KUKA KRL program: MyProgram_091().src

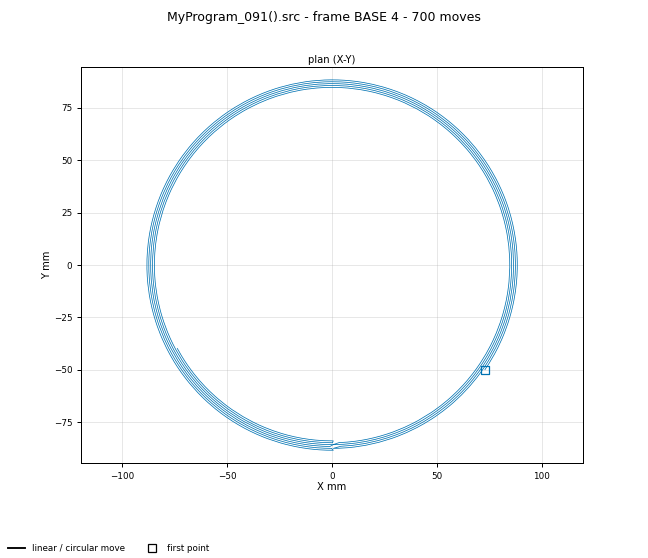
[picture p0: tool path of MyProgram_091().src in frame BASE 4, 700 of 700 moves have a stored position in this frame; points joined in program order, loops and branches not executed]
&ACCESS RVP
&REL 1
&PARAM TEMPLATE = C:\KRC\Roboter\Template\vorgabe
&PARAM EDITMASK = *
DEF MyProgram_091()
; ---- Setting reference (Base) ----
$BASE = BASE_DATA[4]

; --------------------------
; ---- Setting tool (TCP) ----
$TOOL = TOOL_DATA[3]
; --------------------------

$VEL.CP = VEL_APROX_PRINT
Startdeposition()
$VEL.CP = VEL_PRINT
LIN {X 72.876,Y -49.889,Z 87,A -38.6628,B 24.9212,C -2.0494,E1 25.1329,E2 483.5993} C_DIS
LIN {X 74.7508,Y -47.0321,Z 87,A -36.5976,B 24.9212,C -2.0503,E1 25.136,E2 481.5424} C_DIS
LIN {X 77.4491,Y -42.4429,Z 87,A -33.0497,B 24.9201,C -2.0636,E1 25.141,E2 477.9815} C_DIS
LIN {X 79.025,Y -39.4299,Z 87,A -30.5206,B 24.9187,C -2.0816,E1 25.1442,E2 475.4232} C_DIS
LIN {X 80.9108,Y -35.3988,Z 87,A -27.9647,B 24.919,C -2.0785,E1 25.1471,E2 472.8887} C_DIS
LIN {X 82.1401,Y -32.4446,Z 87,A -25.9813,B 24.9187,C -2.0815,E1 25.1492,E2 470.9091} C_DIS
LIN {X 83.9091,Y -27.5504,Z 87,A -22.6052,B 24.9179,C -2.0919,E1 25.1523,E2 467.5274} C_DIS
LIN {X 84.8703,Y -24.4292,Z 87,A -20.491,B 24.9174,C -2.0984,E1 25.154,E2 465.41} C_DIS
LIN {X 85.5175,Y -22.0541,Z 87,A -18.418,B 24.9157,C -2.1205,E1 25.1555,E2 463.2967} C_DIS
LIN {X 86.2783,Y -18.8591,Z 87,A -16.8201,B 24.9167,C -2.1081,E1 25.1564,E2 461.7374} C_DIS
LIN {X 86.7492,Y -16.5591,Z 87,A -15.0502,B 24.9156,C -2.1218,E1 25.1574,E2 459.9455} C_DIS
LIN {X 87.4227,Y -12.5256,Z 87,A -12.6764,B 24.9156,C -2.1203,E1 25.1584,E2 457.5893} C_DIS
LIN {X 87.8803,Y -8.7666,Z 87,A -10.1907,B 24.915,C -2.1292,E1 25.1591,E2 455.0972} C_DIS
LIN {X 88.1529,Y -5.3772,Z 87,A -7.9487,B 24.9143,C -2.1375,E1 25.1596,E2 452.8488} C_DIS
LIN {X 88.2975,Y -1.7856,Z 87,A -5.7756,B 24.9142,C -2.1393,E1 25.1598,E2 450.6844} C_DIS
LIN {X 88.3023,Y 1.525,Z 87,A -3.8298,B 24.9142,C -2.139,E1 25.1598,E2 448.751} C_DIS
LIN {X 88.2492,Y 3.4377,Z 87,A -2.4189,B 24.9134,C -2.149,E1 25.1596,E2 447.3249} C_DIS
LIN {X 88.101,Y 6.1542,Z 87,A -0.5423,B 24.9126,C -2.1586,E1 25.1593,E2 445.4368} C_DIS
LIN {X 87.7851,Y 9.6757,Z 87,A 1.7717,B 24.912,C -2.1666,E1 25.1586,E2 443.1177} C_DIS
LIN {X 87.4539,Y 12.306,Z 87,A 3.3765,B 24.9118,C -2.1679,E1 25.158,E2 441.5192} C_DIS
LIN {X 86.9147,Y 15.667,Z 87,A 6.3248,B 24.9091,C -2.2013,E1 25.1566,E2 438.5094} C_DIS
LIN {X 86.0978,Y 19.6679,Z 87,A 8.2385,B 24.9106,C -2.1831,E1 25.1554,E2 436.6497} C_DIS
LIN {X 85.2224,Y 23.1685,Z 87,A 11.3311,B 24.9078,C -2.217,E1 25.1532,E2 433.4948} C_DIS
LIN {X 84.0146,Y 27.2242,Z 87,A 13.1855,B 24.9098,C -2.1935,E1 25.1517,E2 431.7066} C_DIS
LIN {X 82.9978,Y 30.1827,Z 87,A 14.9428,B 24.9101,C -2.1898,E1 25.15,E2 429.9677} C_DIS
LIN {X 81.9785,Y 32.8537,Z 87,A 17.2118,B 24.9084,C -2.2098,E1 25.1477,E2 427.6642} C_DIS
LIN {X 80.5997,Y 36.1019,Z 87,A 19.3758,B 24.9082,C -2.2119,E1 25.1453,E2 425.507} C_DIS
LIN {X 79.2608,Y 38.9542,Z 87,A 21.315,B 24.9081,C -2.2139,E1 25.143,E2 423.5735} C_DIS
LIN {X 77.959,Y 41.4989,Z 87,A 23.2226,B 24.9075,C -2.2209,E1 25.1405,E2 421.6595} C_DIS
LIN {X 76.1764,Y 44.6862,Z 87,A 25.6641,B 24.9067,C -2.2298,E1 25.1371,E2 419.2097} C_DIS
LIN {X 74.6097,Y 47.2577,Z 87,A 27.6005,B 24.9064,C -2.2342,E1 25.1342,E2 417.2726} C_DIS
LIN {X 72.7642,Y 50.0518,Z 87,A 29.7426,B 24.906,C -2.2387,E1 25.1309,E2 415.1305} C_DIS
LIN {X 70.4422,Y 53.269,Z 87,A 32.3068,B 24.9055,C -2.2447,E1 25.1267,E2 412.5645} C_DIS
LIN {X 68.1897,Y 56.1245,Z 87,A 34.6943,B 24.9049,C -2.2512,E1 25.1225,E2 410.1727} C_DIS
LIN {X 64.9745,Y 59.816,Z 87,A 37.8698,B 24.9043,C -2.2584,E1 25.1166,E2 406.9945} C_DIS
LIN {X 62.6446,Y 62.2522,Z 87,A 39.9936,B 24.9041,C -2.2609,E1 25.1124,E2 404.8738} C_DIS
LIN {X 60.3809,Y 64.4499,Z 87,A 42.1613,B 24.9034,C -2.2692,E1 25.108,E2 402.6953} C_DIS
LIN {X 57.7117,Y 66.8523,Z 87,A 44.4118,B 24.9032,C -2.2711,E1 25.1033,E2 400.4494} C_DIS
LIN {X 55.9301,Y 68.3492,Z 87,A 46.0715,B 24.9026,C -2.279,E1 25.0997,E2 398.7771} C_DIS
LIN {X 52.7405,Y 70.8393,Z 87,A 48.5236,B 24.9026,C -2.2778,E1 25.0943,E2 396.3369} C_DIS
LIN {X 49.8742,Y 72.886,Z 87,A 50.7541,B 24.9025,C -2.2797,E1 25.0892,E2 394.1095} C_DIS
LIN {X 47.2166,Y 74.6354,Z 87,A 52.8049,B 24.9023,C -2.2825,E1 25.0844,E2 392.0588} C_DIS
LIN {X 44.6136,Y 76.2193,Z 87,A 54.8992,B 24.9017,C -2.2894,E1 25.0793,E2 389.9547} C_DIS
LIN {X 40.7584,Y 78.349,Z 87,A 57.6799,B 24.9016,C -2.2906,E1 25.0725,E2 387.179} C_DIS
LIN {X 37.7561,Y 79.8391,Z 87,A 59.8219,B 24.9014,C -2.2922,E1 25.0671,E2 385.0389} C_DIS
LIN {X 34.8344,Y 81.1568,Z 87,A 61.9798,B 24.901,C -2.2971,E1 25.0616,E2 382.8748} C_DIS
LIN {X 31.3951,Y 82.5468,Z 87,A 64.2661,B 24.9011,C -2.2954,E1 25.0556,E2 380.5973} C_DIS
LIN {X 27.7885,Y 83.8309,Z 87,A 66.9063,B 24.9005,C -2.3027,E1 25.0486,E2 377.945} C_DIS
LIN {X 24.1511,Y 84.9491,Z 87,A 69.3497,B 24.9005,C -2.3037,E1 25.0421,E2 375.5036} C_DIS
LIN {X 19.3333,Y 86.1749,Z 87,A 72.7743,B 24.8997,C -2.3119,E1 25.0328,E2 372.0643} C_DIS
LIN {X 15.0004,Y 87.0333,Z 87,A 75.3209,B 24.9005,C -2.3027,E1 25.0258,E2 369.5426} C_DIS
LIN {X 11.7786,Y 87.5275,Z 87,A 77.488,B 24.9003,C -2.3049,E1 25.0198,E2 367.3721} C_DIS
LIN {X 8.3793,Y 87.9174,Z 87,A 79.6385,B 24.9005,C -2.303,E1 25.0139,E2 365.2275} C_DIS
LIN {X 5.8507,Y 88.1215,Z 87,A 81.1313,B 24.9009,C -2.2981,E1 25.0098,E2 363.7469} C_DIS
LIN {X 2.8316,Y 88.2701,Z 87,A 83.2135,B 24.9006,C -2.3019,E1 25.0039,E2 361.6564} C_DIS
LIN {X -0.4871,Y 88.3141,Z 87,A 85.3405,B 24.9006,C -2.3007,E1 24.998,E2 359.5324} C_DIS
LIN {X -3.58,Y 88.2431,Z 87,A 87.5251,B 24.9003,C -2.3057,E1 24.9919,E2 357.3356} C_DIS
LIN {X -9.587,Y 87.7944,Z 87,A 91.3179,B 24.9007,C -2.3002,E1 24.9814,E2 353.5541} C_DIS
LIN {X -12.8181,Y 87.3812,Z 87,A 93.176,B 24.9015,C -2.2909,E1 24.9763,E2 351.7167} C_DIS
LIN {X -19.1362,Y 86.2179,Z 87,A 98.0168,B 24.9,C -2.3085,E1 24.9629,E2 346.8286} C_DIS
LIN {X -24.8016,Y 84.762,Z 87,A 101.1149,B 24.9022,C -2.283,E1 24.9547,E2 343.7865} C_DIS
LIN {X -27.1803,Y 84.0288,Z 87,A 102.9141,B 24.9019,C -2.2868,E1 24.9498,E2 341.975} C_DIS
LIN {X -30.117,Y 83.0217,Z 87,A 104.987,B 24.9019,C -2.2861,E1 24.9444,E2 339.8997} C_DIS
LIN {X -33.1255,Y 81.8679,Z 87,A 107.1485,B 24.902,C -2.2855,E1 24.9387,E2 337.735} C_DIS
LIN {X -36.3766,Y 80.4759,Z 87,A 109.4796,B 24.9022,C -2.2832,E1 24.9328,E2 335.4037} C_DIS
LIN {X -39.1194,Y 79.1789,Z 87,A 111.3587,B 24.9027,C -2.2774,E1 24.9281,E2 333.5336} C_DIS
LIN {X -41.9795,Y 77.7004,Z 87,A 113.3448,B 24.9033,C -2.2709,E1 24.9232,E2 331.5577} C_DIS
LIN {X -46.5097,Y 75.0771,Z 87,A 116.9653,B 24.9033,C -2.2715,E1 24.9145,E2 327.9247} C_DIS
LIN {X -49.4678,Y 73.1612,Z 87,A 119.2238,B 24.9036,C -2.2663,E1 24.9092,E2 325.6712} C_DIS
LIN {X -52.1803,Y 71.2519,Z 87,A 121.7484,B 24.9031,C -2.2731,E1 24.9035,E2 323.1215} C_DIS
LIN {X -56.1307,Y 68.1845,Z 87,A 124.6939,B 24.9044,C -2.2571,E1 24.8971,E2 320.2031} C_DIS
LIN {X -58.7959,Y 65.899,Z 87,A 126.8822,B 24.9051,C -2.2494,E1 24.8925,E2 318.0248} C_DIS
LIN {X -61.1916,Y 63.6807,Z 87,A 129.2287,B 24.9049,C -2.2512,E1 24.8877,E2 315.6642} C_DIS
LIN {X -63.993,Y 60.8667,Z 87,A 131.6694,B 24.9058,C -2.2409,E1 24.883,E2 313.2375} C_DIS
LIN {X -66.1895,Y 58.4706,Z 87,A 133.8713,B 24.906,C -2.2384,E1 24.8789,E2 311.0319} C_DIS
LIN {X -68.3105,Y 55.9778,Z 87,A 136.0783,B 24.9063,C -2.2353,E1 24.8749,E2 308.8219} C_DIS
LIN {X -71.2925,Y 52.1248,Z 87,A 139.5827,B 24.9061,C -2.237,E1 24.869,E2 305.2966} C_DIS
LIN {X -73.1619,Y 49.4667,Z 87,A 141.0522,B 24.9082,C -2.2125,E1 24.8668,E2 303.8784} C_DIS
LIN {X -75.9695,Y 45.0363,Z 87,A 144.5868,B 24.9087,C -2.2067,E1 24.8616,E2 300.3396} C_DIS
LIN {X -77.3872,Y 42.557,Z 87,A 146.5252,B 24.9089,C -2.2038,E1 24.8589,E2 298.3979} C_DIS
LIN {X -78.8169,Y 39.8455,Z 87,A 148.6496,B 24.9091,C -2.202,E1 24.8562,E2 296.2666} C_DIS
LIN {X -80.4836,Y 36.3595,Z 87,A 150.9735,B 24.9101,C -2.1892,E1 24.8535,E2 293.9605} C_DIS
LIN {X -81.7261,Y 33.4739,Z 87,A 153.0561,B 24.9105,C -2.1843,E1 24.8512,E2 291.878} C_DIS
LIN {X -82.8825,Y 30.4988,Z 87,A 155.1598,B 24.9109,C -2.1789,E1 24.8492,E2 289.7753} C_DIS
LIN {X -83.9638,Y 27.3812,Z 87,A 157.4119,B 24.9112,C -2.1755,E1 24.8472,E2 287.5185} C_DIS
LIN {X -84.9579,Y 24.1201,Z 87,A 159.5991,B 24.9118,C -2.1679,E1 24.8454,E2 285.3368} C_DIS
LIN {X -85.7975,Y 20.9382,Z 87,A 161.6195,B 24.9127,C -2.1579,E1 24.8441,E2 283.3285} C_DIS
LIN {X -86.4497,Y 18.0599,Z 87,A 163.6354,B 24.9129,C -2.1547,E1 24.8429,E2 281.3083} C_DIS
LIN {X -87.0374,Y 14.9757,Z 87,A 165.6786,B 24.9134,C -2.1484,E1 24.8419,E2 279.268} C_DIS
LIN {X -87.5816,Y 11.3616,Z 87,A 168.9039,B 24.912,C -2.1657,E1 24.8407,E2 275.9822} C_DIS
LIN {X -88.0383,Y 6.9906,Z 87,A 171.1962,B 24.9141,C -2.1403,E1 24.8401,E2 273.7369} C_DIS
LIN {X -88.2709,Y 2.807,Z 87,A 173.5689,B 24.9156,C -2.1216,E1 24.8398,E2 271.3945} C_DIS
LIN {X -88.2983,Y -1.7412,Z 87,A 176.7792,B 24.9157,C -2.1197,E1 24.8398,E2 268.1695} C_DIS
LIN {X -88.1559,Y -5.3252,Z 87,A 178.975,B 24.9166,C -2.1084,E1 24.8402,E2 265.9872} C_DIS
LIN {X -87.8679,Y -8.8855,Z 87,A -178.2885,B 24.9162,C -2.1133,E1 24.8409,E2 263.2227} C_DIS
LIN {X -87.1817,Y -14.1128,Z 87,A -175.1401,B 24.9177,C -2.0947,E1 24.8422,E2 260.1} C_DIS
LIN {X -86.608,Y -17.2887,Z 87,A -173.0562,B 24.9182,C -2.0879,E1 24.8432,E2 258.02} C_DIS
LIN {X -85.8301,Y -20.8043,Z 87,A -170.8084,B 24.919,C -2.0782,E1 24.8447,E2 255.7821} C_DIS
LIN {X -85.1046,Y -23.6023,Z 87,A -168.8704,B 24.9193,C -2.0743,E1 24.8461,E2 253.8421} C_DIS
LIN {X -84.1569,Y -26.7844,Z 87,A -166.6296,B 24.9196,C -2.0704,E1 24.8479,E2 251.5977} C_DIS
LIN {X -83.3448,Y -29.2106,Z 87,A -164.2506,B 24.9183,C -2.0868,E1 24.8502,E2 249.1663} C_DIS
LIN {X -81.8433,Y -33.186,Z 87,A -162.2766,B 24.9208,C -2.0557,E1 24.8522,E2 247.2554} C_DIS
LIN {X -80.9152,Y -35.3886,Z 87,A -160.3188,B 24.9202,C -2.0632,E1 24.8544,E2 245.2687} C_DIS
LIN {X -79.0112,Y -39.4578,Z 87,A -157.8931,B 24.9219,C -2.0407,E1 24.8573,E2 242.8837} C_DIS
LIN {X -77.5103,Y -42.3301,Z 87,A -155.4738,B 24.9216,C -2.0443,E1 24.8605,E2 240.4428} C_DIS
LIN {X -75.5172,Y -45.7905,Z 87,A -153.1118,B 24.9227,C -2.0307,E1 24.8638,E2 238.1011} C_DIS
LIN {X -73.8148,Y -48.4873,Z 87,A -150.9893,B 24.923,C -2.027,E1 24.867,E2 235.9768} C_DIS
LIN {X -71.9019,Y -51.281,Z 87,A -148.6632,B 24.923,C -2.0254,E1 24.8708,E2 233.643} C_DIS
LIN {X -69.5864,Y -54.3836,Z 87,A -146.2279,B 24.9237,C -2.017,E1 24.8749,E2 231.2161} C_DIS
LIN {X -68.083,Y -56.2528,Z 87,A -144.2851,B 24.9231,C -2.0251,E1 24.8784,E2 229.2452} C_DIS
LIN {X -64.0638,Y -60.7914,Z 87,A -140.5474,B 24.9242,C -2.0104,E1 24.8854,E2 225.5258} C_DIS
LIN {X -61.2434,Y -63.6307,Z 87,A -138.2242,B 24.9252,C -1.9968,E1 24.8899,E2 223.2254} C_DIS
LIN {X -59.1443,Y -65.5871,Z 87,A -136.313,B 24.9254,C -1.9945,E1 24.8939,E2 221.3117} C_DIS
LIN {X -55.4752,Y -68.7179,Z 87,A -133.0922,B 24.9256,C -1.9914,E1 24.9008,E2 218.0859} C_DIS
LIN {X -52.8784,Y -70.7356,Z 87,A -130.9123,B 24.9258,C -1.9891,E1 24.9056,E2 215.9037} C_DIS
LIN {X -50.2741,Y -72.6096,Z 87,A -128.825,B 24.9261,C -1.9858,E1 24.9104,E2 213.817} C_DIS
LIN {X -47.5755,Y -74.4057,Z 87,A -126.707,B 24.9263,C -1.983,E1 24.9154,E2 211.6989} C_DIS
LIN {X -44.9756,Y -76.0053,Z 87,A -124.6208,B 24.9263,C -1.9834,E1 24.9204,E2 209.6053} C_DIS
LIN {X -41.6869,Y -77.8592,Z 87,A -122.2867,B 24.9268,C -1.9766,E1 24.9261,E2 207.2809} C_DIS
LIN {X -38.9012,Y -79.2871,Z 87,A -120.2764,B 24.927,C -1.9734,E1 24.9311,E2 205.2727} C_DIS
LIN {X -36.1322,Y -80.586,Z 87,A -118.266,B 24.927,C -1.972,E1 24.9362,E2 203.2607} C_DIS
LIN {X -32.7878,Y -82.0053,Z 87,A -115.8818,B 24.9272,C -1.9705,E1 24.9424,E2 200.8747} C_DIS
LIN {X -30.3038,Y -82.9536,Z 87,A -113.7469,B 24.9263,C -1.982,E1 24.948,E2 198.7082} C_DIS
LIN {X -24.4184,Y -84.8733,Z 87,A -110.1572,B 24.9276,C -1.9654,E1 24.9575,E2 195.1516} C_DIS
LIN {X -22.1968,Y -85.4808,Z 87,A -108.4317,B 24.9271,C -1.972,E1 24.9622,E2 193.4081} C_DIS
LIN {X -18.1313,Y -86.435,Z 87,A -106.0112,B 24.9279,C -1.9614,E1 24.9688,E2 191.0096} C_DIS
LIN {X -15.1651,Y -87.0049,Z 87,A -103.9211,B 24.9276,C -1.9649,E1 24.9745,E2 188.909} C_DIS
LIN {X -11.645,Y -87.5448,Z 87,A -101.7389,B 24.928,C -1.9603,E1 24.9805,E2 186.736} C_DIS
LIN {X -9.0148,Y -87.8543,Z 87,A -100.1645,B 24.9283,C -1.9554,E1 24.9849,E2 185.1722} C_DIS
LIN {X -6.1629,Y -88.1004,Z 87,A -98.1033,B 24.9278,C -1.962,E1 24.9907,E2 183.0945} C_DIS
LIN {X -2.6223,Y -88.2765,Z 87,A -95.8044,B 24.9278,C -1.9622,E1 24.9971,E2 180.7946} C_DIS
LIN {X 0.5878,Y -88.3126,Z 87,A -94.072,B 24.9286,C -1.9512,E1 25.0019,E2 179.0883} C_DIS
Enddeposition()
LIN {X 0.5878,Y -88.3126,Z 87,A -94.072,B 24.9286,C -1.9512,E1 25.0019,E2 179.0883} C_DIS
Startdeposition()
$VEL.CP = VEL_PRINT
LIN {X -0.2815,Y -87.4214,Z 87,A -95.3283,B 24.9291,C -1.9446,E1 24.9983,E2 180.3603} C_DIS
LIN {X -3.6833,Y -87.3438,Z 87,A -97.4905,B 24.929,C -1.9464,E1 24.9923,E2 182.5184} C_DIS
LIN {X -7.3441,Y -87.113,Z 87,A -100.0671,B 24.9294,C -1.941,E1 24.9851,E2 185.1089} C_DIS
LIN {X -10.6188,Y -86.7753,Z 87,A -102.1476,B 24.9292,C -1.9437,E1 24.9793,E2 187.1844} C_DIS
LIN {X -13.9854,Y -86.2966,Z 87,A -104.6701,B 24.9298,C -1.9351,E1 24.9723,E2 189.7295} C_DIS
LIN {X -18.097,Y -85.5294,Z 87,A -107.3335,B 24.9295,C -1.9386,E1 24.965,E2 192.3876} C_DIS
LIN {X -22.0017,Y -84.6079,Z 87,A -109.8167,B 24.9291,C -1.9446,E1 24.9583,E2 194.86} C_DIS
LIN {X -26.6799,Y -83.2511,Z 87,A -113.3252,B 24.9296,C -1.9372,E1 24.9489,E2 198.3922} C_DIS
LIN {X -30.4817,Y -81.9368,Z 87,A -115.7071,B 24.9289,C -1.9472,E1 24.9427,E2 200.755} C_DIS
LIN {X -35.5927,Y -79.8486,Z 87,A -118.9086,B 24.9277,C -1.9636,E1 24.9345,E2 203.9248} C_DIS
LIN {X -39.0234,Y -78.2287,Z 87,A -121.728,B 24.9282,C -1.9565,E1 24.9273,E2 206.7684} C_DIS
LIN {X -44.0876,Y -75.4917,Z 87,A -125.2495,B 24.9273,C -1.9691,E1 24.9188,E2 210.27} C_DIS
LIN {X -48.2363,Y -72.9095,Z 87,A -128.7326,B 24.9276,C -1.9656,E1 24.9105,E2 213.7726} C_DIS
LIN {X -50.9762,Y -71.0211,Z 87,A -130.8701,B 24.9272,C -1.9705,E1 24.9056,E2 215.9058} C_DIS
LIN {X -53.7697,Y -68.9313,Z 87,A -133.2694,B 24.9272,C -1.9711,E1 24.9003,E2 218.3122} C_DIS
LIN {X -57.5317,Y -65.8226,Z 87,A -136.2874,B 24.9263,C -1.9825,E1 24.8939,E2 221.3147} C_DIS
LIN {X -59.9471,Y -63.6306,Z 87,A -138.5032,B 24.9262,C -1.9845,E1 24.8893,E2 223.5348} C_DIS
LIN {X -62.283,Y -61.3462,Z 87,A -140.4609,B 24.9254,C -1.9944,E1 24.8855,E2 225.4772} C_DIS
LIN {X -64.2029,Y -59.3343,Z 87,A -143.2591,B 24.9272,C -1.97,E1 24.88,E2 228.3457} C_DIS
LIN {X -66.928,Y -56.2439,Z 87,A -145.2973,B 24.9254,C -1.9953,E1 24.8764,E2 230.3331} C_DIS
LIN {X -69.0342,Y -53.6369,Z 87,A -147.4346,B 24.9248,C -2.0022,E1 24.8727,E2 232.4639} C_DIS
LIN {X -71.7597,Y -49.9304,Z 87,A -150.3799,B 24.9241,C -2.0116,E1 24.8679,E2 235.401} C_DIS
LIN {X -73.529,Y -47.2864,Z 87,A -152.4797,B 24.9238,C -2.0165,E1 24.8647,E2 237.4997} C_DIS
LIN {X -75.1206,Y -44.7155,Z 87,A -155.034,B 24.9246,C -2.0054,E1 24.861,E2 240.0938} C_DIS
LIN {X -76.7069,Y -41.9362,Z 87,A -156.4886,B 24.9228,C -2.0293,E1 24.8591,E2 241.4988} C_DIS
LIN {X -77.996,Y -39.4872,Z 87,A -158.5283,B 24.9228,C -2.0278,E1 24.8564,E2 243.553} C_DIS
LIN {X -79.9903,Y -35.2731,Z 87,A -161.2883,B 24.9216,C -2.0448,E1 24.8532,E2 246.2876} C_DIS
LIN {X -82.473,Y -28.995,Z 87,A -165.5487,B 24.9202,C -2.0623,E1 24.8489,E2 250.53} C_DIS
LIN {X -83.3285,Y -26.4405,Z 87,A -167.6251,B 24.9205,C -2.0587,E1 24.847,E2 252.627} C_DIS
LIN {X -84.0991,Y -23.8717,Z 87,A -169.5061,B 24.9204,C -2.0605,E1 24.8456,E2 254.5146} C_DIS
LIN {X -84.9072,Y -20.8155,Z 87,A -171.738,B 24.9202,C -2.0623,E1 24.844,E2 256.7551} C_DIS
LIN {X -85.6661,Y -17.4313,Z 87,A -174.0113,B 24.9197,C -2.0693,E1 24.8427,E2 259.0252} C_DIS
LIN {X -86.3301,Y -13.7767,Z 87,A -177.6579,B 24.9217,C -2.0433,E1 24.8411,E2 262.7555} C_DIS
LIN {X -87.0454,Y -8.1,Z 87,A 178.8467,B 24.9203,C -2.0621,E1 24.8401,E2 266.2269} C_DIS
LIN {X -87.3637,Y -3.2192,Z 87,A 175.6459,B 24.9195,C -2.0724,E1 24.8398,E2 269.4224} C_DIS
LIN {X -87.4091,Y 1.474,Z 87,A 173.9242,B 24.9157,C -2.1199,E1 24.8398,E2 271.0412} C_DIS
LIN {X -87.3331,Y 3.934,Z 87,A 171.6616,B 24.9168,C -2.1069,E1 24.8401,E2 273.3485} C_DIS
LIN {X -87.0479,Y 8.0725,Z 87,A 168.765,B 24.9165,C -2.1106,E1 24.8407,E2 276.2535} C_DIS
LIN {X -86.6798,Y 11.3639,Z 87,A 166.5592,B 24.916,C -2.1166,E1 24.8415,E2 278.4583} C_DIS
LIN {X -85.9844,Y 15.789,Z 87,A 164.0337,B 24.9143,C -2.1373,E1 24.8427,E2 280.9493} C_DIS
LIN {X -85.328,Y 19.0211,Z 87,A 161.7929,B 24.914,C -2.1419,E1 24.844,E2 283.1922} C_DIS
LIN {X -84.5943,Y 22.0546,Z 87,A 159.5132,B 24.914,C -2.1419,E1 24.8456,E2 285.4854} C_DIS
LIN {X -83.6246,Y 25.4874,Z 87,A 156.7807,B 24.9143,C -2.1382,E1 24.8478,E2 288.2424} C_DIS
LIN {X -82.495,Y 28.9323,Z 87,A 155.1787,B 24.9119,C -2.1671,E1 24.8492,E2 289.7846} C_DIS
LIN {X -81.5821,Y 31.4182,Z 87,A 153.2073,B 24.912,C -2.1657,E1 24.8511,E2 291.7702} C_DIS
LIN {X -80.3185,Y 34.5202,Z 87,A 151.0087,B 24.9115,C -2.1723,E1 24.8535,E2 293.9655} C_DIS
LIN {X -78.2485,Y 38.9835,Z 87,A 147.8629,B 24.9105,C -2.1841,E1 24.8573,E2 297.1002} C_DIS
LIN {X -76.8564,Y 41.6606,Z 87,A 145.8722,B 24.9101,C -2.1895,E1 24.8598,E2 299.0886} C_DIS
LIN {X -75.0813,Y 44.7821,Z 87,A 142.9305,B 24.9109,C -2.1797,E1 24.8641,E2 302.0689} C_DIS
LIN {X -73.2991,Y 47.6445,Z 87,A 141.3474,B 24.9089,C -2.2035,E1 24.8664,E2 303.6033} C_DIS
LIN {X -70.2212,Y 52.0747,Z 87,A 137.8441,B 24.9081,C -2.214,E1 24.872,E2 307.0986} C_DIS
LIN {X -66.9526,Y 56.2144,Z 87,A 134.2956,B 24.9075,C -2.2204,E1 24.8782,E2 310.6484} C_DIS
LIN {X -64.9688,Y 58.4947,Z 87,A 131.55,B 24.9089,C -2.2037,E1 24.8834,E2 313.4461} C_DIS
LIN {X -62.3923,Y 61.2355,Z 87,A 129.1604,B 24.9082,C -2.2118,E1 24.888,E2 315.8266} C_DIS
LIN {X -59.9315,Y 63.6453,Z 87,A 127.869,B 24.9055,C -2.2448,E1 24.8905,E2 317.0448} C_DIS
LIN {X -58.2079,Y 65.2255,Z 87,A 125.9205,B 24.9062,C -2.2363,E1 24.8946,E2 319.0214} C_DIS
LIN {X -54.3965,Y 68.4368,Z 87,A 121.878,B 24.9075,C -2.2212,E1 24.9034,E2 323.1152} C_DIS
LIN {X -51.1215,Y 70.9172,Z 87,A 120.0023,B 24.905,C -2.2502,E1 24.9075,E2 324.9285} C_DIS
LIN {X -46.6715,Y 73.922,Z 87,A 116.4269,B 24.9046,C -2.2553,E1 24.9159,E2 328.5034} C_DIS
LIN {X -42.8092,Y 76.2229,Z 87,A 113.7539,B 24.9034,C -2.2686,E1 24.9222,E2 331.1528} C_DIS
LIN {X -40.0064,Y 77.7307,Z 87,A 111.3985,B 24.9038,C -2.2641,E1 24.9281,E2 333.5254} C_DIS
LIN {X -37.477,Y 78.9821,Z 87,A 109.4452,B 24.9038,C -2.2639,E1 24.933,E2 335.4842} C_DIS
LIN {X -34.3677,Y 80.3839,Z 87,A 107.1756,B 24.9037,C -2.2662,E1 24.9388,E2 337.7538} C_DIS
LIN {X -31.2164,Y 81.6585,Z 87,A 105.0576,B 24.9031,C -2.2725,E1 24.9443,E2 339.8615} C_DIS
LIN {X -28.3477,Y 82.6989,Z 87,A 102.6475,B 24.9039,C -2.2628,E1 24.9507,E2 342.2993} C_DIS
LIN {X -24.2511,Y 83.9916,Z 87,A 99.118,B 24.9055,C -2.2447,E1 24.9603,E2 345.8777} C_DIS
LIN {X -19.3296,Y 85.2584,Z 87,A 97.0433,B 24.902,C -2.2853,E1 24.9657,E2 347.8585} C_DIS
LIN {X -13.4502,Y 86.3806,Z 87,A 93.3511,B 24.9012,C -2.2953,E1 24.9758,E2 351.5308} C_DIS
LIN {X -8.9325,Y 86.9641,Z 87,A 89.8061,B 24.9025,C -2.28,E1 24.9857,E2 355.1148} C_DIS
LIN {X -3.5801,Y 87.3483,Z 87,A 86.4883,B 24.9018,C -2.2875,E1 24.9949,E2 358.4159} C_DIS
LIN {X -0.5659,Y 87.4196,Z 87,A 84.4511,B 24.902,C -2.2861,E1 25.0006,E2 360.4565} C_DIS
LIN {X 3.8734,Y 87.3357,Z 87,A 81.3014,B 24.9026,C -2.2789,E1 25.0094,E2 363.6225} C_DIS
LIN {X 6.8273,Y 87.1546,Z 87,A 79.5609,B 24.902,C -2.285,E1 25.0142,E2 365.3477} C_DIS
LIN {X 10.4424,Y 86.796,Z 87,A 76.7873,B 24.9031,C -2.2724,E1 25.022,E2 368.1493} C_DIS
LIN {X 14.5641,Y 86.1999,Z 87,A 74.4677,B 24.9021,C -2.2844,E1 25.0283,E2 370.4381} C_DIS
LIN {X 18.4518,Y 85.4522,Z 87,A 72.2307,B 24.9012,C -2.2946,E1 25.0344,E2 372.6482} C_DIS
LIN {X 21.2995,Y 84.7873,Z 87,A 69.4478,B 24.9037,C -2.2661,E1 25.0421,E2 375.4948} C_DIS
LIN {X 24.5101,Y 83.916,Z 87,A 67.4811,B 24.9032,C -2.2713,E1 25.0473,E2 377.4458} C_DIS
LIN {X 27.4048,Y 83.0166,Z 87,A 65.6436,B 24.9029,C -2.2744,E1 25.0522,E2 379.2724} C_DIS
LIN {X 32.354,Y 81.2152,Z 87,A 62.3496,B 24.9028,C -2.2763,E1 25.0607,E2 382.555} C_DIS
LIN {X 35.4332,Y 79.9205,Z 87,A 60.0848,B 24.9032,C -2.2715,E1 25.0666,E2 384.8258} C_DIS
LIN {X 38.6942,Y 78.3919,Z 87,A 57.2706,B 24.9047,C -2.254,E1 25.0737,E2 387.6739} C_DIS
LIN {X 41.7201,Y 76.8241,Z 87,A 55.8727,B 24.9026,C -2.2781,E1 25.077,E2 389.0107} C_DIS
LIN {X 44.9466,Y 74.984,Z 87,A 53.0207,B 24.9041,C -2.2609,E1 25.084,E2 391.8947} C_DIS
LIN {X 47.9452,Y 73.1014,Z 87,A 50.8877,B 24.9039,C -2.2635,E1 25.089,E2 394.0147} C_DIS
LIN {X 50.4236,Y 71.4154,Z 87,A 48.5765,B 24.9051,C -2.2488,E1 25.0943,E2 396.3527} C_DIS
LIN {X 55.2652,Y 67.7373,Z 87,A 44.9135,B 24.9048,C -2.2523,E1 25.1023,E2 399.994} C_DIS
LIN {X 57.8195,Y 65.5713,Z 87,A 41.9618,B 24.9073,C -2.223,E1 25.1087,E2 403.0034} C_DIS
LIN {X 60.8637,Y 62.755,Z 87,A 40.141,B 24.9053,C -2.2471,E1 25.1122,E2 404.7595} C_DIS
LIN {X 64.2879,Y 59.242,Z 87,A 36.4786,B 24.9071,C -2.2252,E1 25.1193,E2 408.4579} C_DIS
LIN {X 67.4182,Y 55.6541,Z 87,A 33.521,B 24.9073,C -2.2235,E1 25.1247,E2 411.4061} C_DIS
LIN {X 71.2697,Y 50.6277,Z 87,A 30.0504,B 24.9062,C -2.2364,E1 25.1304,E2 414.8296} C_DIS
LIN {X 73.2335,Y 47.7448,Z 87,A 27.3116,B 24.908,C -2.2152,E1 25.1347,E2 417.605} C_DIS
LIN {X 74.857,Y 45.1555,Z 87,A 25.342,B 24.9083,C -2.2111,E1 25.1376,E2 419.5742} C_DIS
LIN {X 77.5189,Y 40.4162,Z 87,A 21.964,B 24.9086,C -2.2078,E1 25.1422,E2 422.9425} C_DIS
LIN {X 78.7383,Y 37.9843,Z 87,A 20.0645,B 24.9093,C -2.1988,E1 25.1445,E2 424.853} C_DIS
LIN {X 80.0936,Y 35.0361,Z 87,A 17.926,B 24.9098,C -2.1924,E1 25.147,E2 426.995} C_DIS
LIN {X 81.8788,Y 30.6347,Z 87,A 14.983,B 24.9101,C -2.1892,E1 25.15,E2 429.9292} C_DIS
LIN {X 82.7822,Y 28.1006,Z 87,A 13.1231,B 24.9108,C -2.1807,E1 25.1517,E2 431.7988} C_DIS
LIN {X 84.5719,Y 22.1387,Z 87,A 9.3093,B 24.9111,C -2.1776,E1 25.1547,E2 435.5981} C_DIS
LIN {X 85.2278,Y 19.4622,Z 87,A 6.4509,B 24.9144,C -2.1358,E1 25.1566,E2 438.5386} C_DIS
LIN {X 86.0495,Y 15.427,Z 87,A 4.7069,B 24.9125,C -2.1603,E1 25.1575,E2 440.2146} C_DIS
LIN {X 86.6597,Y 11.5193,Z 87,A 2.1927,B 24.9129,C -2.1549,E1 25.1585,E2 442.7267} C_DIS
LIN {X 86.9723,Y 8.8543,Z 87,A 0.2169,B 24.914,C -2.1418,E1 25.1591,E2 444.7217} C_DIS
LIN {X 87.2333,Y 5.7348,Z 87,A -1.9873,B 24.9149,C -2.13,E1 25.1596,E2 446.9408} C_DIS
LIN {X 87.4088,Y 1.4931,Z 87,A -4.3291,B 24.9144,C -2.1364,E1 25.1598,E2 449.2534} C_DIS
LIN {X 87.417,Y -1.0134,Z 87,A -6.3322,B 24.9158,C -2.1186,E1 25.1598,E2 451.2866} C_DIS
LIN {X 87.31,Y -4.4298,Z 87,A -8.6604,B 24.9166,C -2.1084,E1 25.1595,E2 453.6251} C_DIS
LIN {X 86.8595,Y -9.9002,Z 87,A -11.6931,B 24.916,C -2.1165,E1 25.1587,E2 456.6206} C_DIS
LIN {X 86.5616,Y -12.2314,Z 87,A -14.4541,B 24.9197,C -2.0693,E1 25.1576,E2 459.4768} C_DIS
LIN {X 85.7946,Y -16.789,Z 87,A -16.2617,B 24.9171,C -2.1019,E1 25.1567,E2 461.1969} C_DIS
LIN {X 84.9309,Y -20.7183,Z 87,A -19.3153,B 24.9189,C -2.079,E1 25.1548,E2 464.2868} C_DIS
LIN {X 84.2168,Y -23.4561,Z 87,A -21.7567,B 24.921,C -2.0529,E1 25.153,E2 466.7758} C_DIS
LIN {X 83.0323,Y -27.3563,Z 87,A -24,B 24.9205,C -2.0593,E1 25.151,E2 468.9912} C_DIS
LIN {X 81.466,Y -31.7154,Z 87,A -26.3567,B 24.9194,C -2.0736,E1 25.1488,E2 471.3011} C_DIS
LIN {X 80.139,Y -34.932,Z 87,A -28.8975,B 24.9206,C -2.0576,E1 25.146,E2 473.8657} C_DIS
LIN {X 78.0172,Y -39.4457,Z 87,A -31.9394,B 24.9208,C -2.0557,E1 25.1424,E2 476.8957} C_DIS
LIN {X 74.9049,Y -45.0766,Z 87,A -36.6981,B 24.9231,C -2.0248,E1 25.1358,E2 481.7027} C_DIS
LIN {X 72.868,Y -48.2991,Z 87,A -38.9414,B 24.923,C -2.0266,E1 25.1324,E2 483.9305} C_DIS
LIN {X 70.9144,Y -51.1257,Z 87,A -41.2551,B 24.9236,C -2.0182,E1 25.1286,E2 486.2526} C_DIS
LIN {X 68.9171,Y -53.7887,Z 87,A -43.113,B 24.9232,C -2.0235,E1 25.1255,E2 488.0893} C_DIS
LIN {X 65.5149,Y -57.884,Z 87,A -46.5556,B 24.9238,C -2.0161,E1 25.1194,E2 491.5337} C_DIS
LIN {X 61.7017,Y -61.9318,Z 87,A -51.4983,B 24.9277,C -1.9632,E1 25.1095,E2 496.5802} C_DIS
LIN {X 57.8191,Y -65.5716,Z 87,A -53.608,B 24.9249,C -2.0016,E1 25.1054,E2 498.5906} C_DIS
LIN {X 56.135,Y -67.0186,Z 87,A -55.5734,B 24.9264,C -1.981,E1 25.1011,E2 500.597} C_DIS
LIN {X 52.7751,Y -69.6948,Z 87,A -58.9401,B 24.9282,C -1.9566,E1 25.0935,E2 504.0092} C_DIS
LIN {X 49.209,Y -72.2567,Z 87,A -60.6143,B 24.9257,C -1.9912,E1 25.0899,E2 505.5959} C_DIS
LIN {X 47.3153,Y -73.5105,Z 87,A -62.3995,B 24.9266,C -1.9782,E1 25.0856,E2 507.4058} C_DIS
LIN {X 43.9616,Y -75.5652,Z 87,A -65.7576,B 24.9289,C -1.9475,E1 25.0774,E2 510.8263} C_DIS
LIN {X 40.4161,Y -77.5188,Z 87,A -67.485,B 24.927,C -1.9737,E1 25.0733,E2 512.4866} C_DIS
LIN {X 35.5789,Y -79.8548,Z 87,A -71.5174,B 24.9286,C -1.9512,E1 25.063,E2 516.562} C_DIS
LIN {X 31.2837,Y -81.6331,Z 87,A -74.1271,B 24.9279,C -1.9614,E1 25.0563,E2 519.1418} C_DIS
LIN {X 28.548,Y -82.6299,Z 87,A -76.1737,B 24.9284,C -1.9544,E1 25.0509,E2 521.2009} C_DIS
LIN {X 22.3783,Y -84.5098,Z 87,A -81.7986,B 24.932,C -1.9047,E1 25.0355,E2 526.9342} C_DIS
LIN {X 16.0654,Y -85.9339,Z 87,A -84.4091,B 24.9285,C -1.9534,E1 25.0287,E2 529.4261} C_DIS
LIN {X 10.6508,Y -86.7716,Z 87,A -88.1146,B 24.9289,C -1.9471,E1 25.0184,E2 533.143} C_DIS
LIN {X 7.6369,Y -87.0882,Z 87,A -90.2414,B 24.9293,C -1.9416,E1 25.0125,E2 535.2817} C_DIS
LIN {X 3.29,Y -87.3603,Z 87,A -93.1733,B 24.9296,C -1.938,E1 25.0043,E2 538.2211} C_DIS
LIN {X 0.5848,Y -87.4184,Z 87,A -94.4306,B 24.9284,C -1.954,E1 25.0009,E2 539.4402} C_DIS
Enddeposition()
LIN {X 0.5848,Y -87.4184,Z 87,A -94.4306,B 24.9284,C -1.954,E1 25.0009,E2 539.4402} C_DIS
Startdeposition()
$VEL.CP = VEL_PRINT
LIN {X 4.0647,Y -86.4324,Z 87,A -91.6323,B 24.926,C -1.9861,E1 25.0089,E2 536.5664} C_DIS
LIN {X 9.8831,Y -85.9614,Z 87,A -87.2077,B 24.9245,C -2.0062,E1 25.0213,E2 532.0966} C_DIS
LIN {X 15.9355,Y -85.0485,Z 87,A -83.8095,B 24.9259,C -1.9878,E1 25.0306,E2 528.7455} C_DIS
LIN {X 21.7813,Y -83.7415,Z 87,A -79.7028,B 24.9253,C -1.9961,E1 25.0418,E2 524.6249} C_DIS
LIN {X 26.6653,Y -82.3162,Z 87,A -76.0571,B 24.9243,C -2.0091,E1 25.0516,E2 520.9549} C_DIS
LIN {X 30.458,Y -80.9898,Z 87,A -73.9788,B 24.9255,C -1.9932,E1 25.0569,E2 518.9183} C_DIS
LIN {X 33.7629,Y -79.6685,Z 87,A -71.2211,B 24.9243,C -2.0099,E1 25.0641,E2 516.1275} C_DIS
LIN {X 37.866,Y -77.8033,Z 87,A -68.1165,B 24.9236,C -2.0186,E1 25.072,E2 513.0105} C_DIS
LIN {X 40.3214,Y -76.5584,Z 87,A -66.1253,B 24.9229,C -2.0273,E1 25.077,E2 511.004} C_DIS
LIN {X 43.7699,Y -74.6411,Z 87,A -63.4486,B 24.9224,C -2.0342,E1 25.0835,E2 508.3192} C_DIS
LIN {X 47.7974,Y -72.128,Z 87,A -60.9273,B 24.9236,C -2.0191,E1 25.0893,E2 505.8418} C_DIS
LIN {X 50.8791,Y -69.9886,Z 87,A -57.9425,B 24.9219,C -2.0412,E1 25.0962,E2 502.8151} C_DIS
LIN {X 54.4321,Y -67.2618,Z 87,A -55.1108,B 24.9217,C -2.043,E1 25.1024,E2 499.9897} C_DIS
LIN {X 57.1812,Y -64.9418,Z 87,A -52.18,B 24.9199,C -2.0673,E1 25.1086,E2 497.0129} C_DIS
LIN {X 60.1656,Y -62.1863,Z 87,A -50.3938,B 24.9218,C -2.0426,E1 25.1121,E2 495.2926} C_DIS
LIN {X 61.9673,Y -60.391,Z 87,A -48.142,B 24.9199,C -2.0662,E1 25.1166,E2 492.9945} C_DIS
LIN {X 64.8567,Y -57.2785,Z 87,A -45.2354,B 24.9191,C -2.0766,E1 25.122,E2 490.0764} C_DIS
LIN {X 67.0422,Y -54.7031,Z 87,A -43.4765,B 24.92,C -2.0659,E1 25.1251,E2 488.351} C_DIS
LIN {X 70.0006,Y -50.8615,Z 87,A -40.3413,B 24.9195,C -2.0719,E1 25.1303,E2 485.2165} C_DIS
LIN {X 71.9918,Y -48.0039,Z 87,A -38.2994,B 24.9197,C -2.0691,E1 25.1335,E2 483.1912} C_DIS
LIN {X 74.38,Y -44.2116,Z 87,A -35.4935,B 24.9195,C -2.0719,E1 25.1377,E2 480.393} C_DIS
LIN {X 76.7665,Y -39.9261,Z 87,A -31.8606,B 24.9177,C -2.0947,E1 25.1426,E2 476.7253} C_DIS
LIN {X 77.8093,Y -37.8535,Z 87,A -30.2707,B 24.9172,C -2.1011,E1 25.1446,E2 475.1288} C_DIS
LIN {X 79.516,Y -34.124,Z 87,A -27.5587,B 24.9166,C -2.1091,E1 25.1476,E2 472.4125} C_DIS
LIN {X 80.5824,Y -31.5198,Z 87,A -25.397,B 24.9153,C -2.1253,E1 25.1499,E2 470.2246} C_DIS
LIN {X 82.1552,Y -27.1622,Z 87,A -22.4681,B 24.9149,C -2.1299,E1 25.1525,E2 467.3014} C_DIS
LIN {X 83.4225,Y -22.9755,Z 87,A -20.0734,B 24.9156,C -2.1214,E1 25.1543,E2 464.9405} C_DIS
LIN {X 84.8623,Y -16.9011,Z 87,A -15.3993,B 24.913,C -2.1534,E1 25.1572,E2 460.218} C_DIS
LIN {X 85.8599,Y -10.7346,Z 87,A -11.8655,B 24.9137,C -2.1455,E1 25.1587,E2 456.7237} C_DIS
LIN {X 86.3033,Y -6.2377,Z 87,A -8.2579,B 24.9111,C -2.1766,E1 25.1596,E2 453.064} C_DIS
LIN {X 86.5143,Y -1.5084,Z 87,A -5.6384,B 24.9118,C -2.1686,E1 25.1598,E2 450.4791} C_DIS
LIN {X 86.5262,Y 0.5859,Z 87,A -3.7422,B 24.91,C -2.1909,E1 25.1598,E2 448.5415} C_DIS
LIN {X 86.2624,Y 6.7689,Z 87,A -0.1597,B 24.9104,C -2.1858,E1 25.1592,E2 444.9922} C_DIS
LIN {X 85.9372,Y 10.0894,Z 87,A 1.6667,B 24.9109,C -2.1795,E1 25.1586,E2 443.1916} C_DIS
LIN {X 85.2273,Y 14.9483,Z 87,A 5.2945,B 24.909,C -2.2027,E1 25.1571,E2 439.5304} C_DIS
LIN {X 84.1562,Y 20.122,Z 87,A 8.7869,B 24.9081,C -2.2132,E1 25.155,E2 436.0335} C_DIS
LIN {X 83.1724,Y 23.8629,Z 87,A 11.5941,B 24.9068,C -2.2295,E1 25.1529,E2 433.2038} C_DIS
LIN {X 81.8781,Y 27.9841,Z 87,A 14.1634,B 24.9068,C -2.2279,E1 25.1507,E2 430.6529} C_DIS
LIN {X 81.0077,Y 30.4107,Z 87,A 16.6963,B 24.904,C -2.2617,E1 25.1481,E2 428.0543} C_DIS
LIN {X 79.3369,Y 34.5348,Z 87,A 18.7165,B 24.9061,C -2.2378,E1 25.146,E2 426.1015} C_DIS
LIN {X 77.7609,Y 37.9542,Z 87,A 21.8655,B 24.9035,C -2.2675,E1 25.1421,E2 422.8994} C_DIS
LIN {X 76.1068,Y 41.1675,Z 87,A 23.8387,B 24.9042,C -2.2595,E1 25.1395,E2 420.9555} C_DIS
LIN {X 74.0419,Y 44.7753,Z 87,A 26.5671,B 24.9037,C -2.2659,E1 25.1357,E2 418.2259} C_DIS
LIN {X 71.9588,Y 48.0539,Z 87,A 28.8842,B 24.9039,C -2.2638,E1 25.1322,E2 415.9255} C_DIS
LIN {X 70.6291,Y 49.9863,Z 87,A 30.8524,B 24.9023,C -2.2818,E1 25.1289,E2 413.9241} C_DIS
LIN {X 67.9003,Y 53.6334,Z 87,A 33.4429,B 24.9029,C -2.2746,E1 25.1246,E2 411.3631} C_DIS
LIN {X 65.5206,Y 56.5184,Z 87,A 36.8645,B 24.8997,C -2.3125,E1 25.1182,E2 407.8673} C_DIS
LIN {X 62.382,Y 59.9625,Z 87,A 39.1269,B 24.9015,C -2.2912,E1 25.114,E2 405.6652} C_DIS
LIN {X 60.023,Y 62.3237,Z 87,A 41.0451,B 24.902,C -2.286,E1 25.1102,E2 403.7673} C_DIS
LIN {X 56.766,Y 65.3044,Z 87,A 44.1657,B 24.9009,C -2.2984,E1 25.1037,E2 400.6299} C_DIS
LIN {X 54.6004,Y 67.1254,Z 87,A 45.9535,B 24.9009,C -2.299,E1 25.0999,E2 398.8473} C_DIS
LIN {X 51.9931,Y 69.1644,Z 87,A 48.0422,B 24.9008,C -2.2995,E1 25.0952,E2 396.7651} C_DIS
LIN {X 49.5006,Y 70.9698,Z 87,A 50.1645,B 24.9003,C -2.3058,E1 25.0904,E2 394.6355} C_DIS
LIN {X 46.6238,Y 72.8919,Z 87,A 52.5052,B 24.8998,C -2.311,E1 25.0849,E2 392.29} C_DIS
LIN {X 41.774,Y 75.777,Z 87,A 56.025,B 24.9,C -2.3092,E1 25.0765,E2 388.7851} C_DIS
LIN {X 39.2892,Y 77.0933,Z 87,A 58.7297,B 24.8973,C -2.3393,E1 25.0696,E2 386.0166} C_DIS
LIN {X 35.7996,Y 78.7748,Z 87,A 60.6009,B 24.8991,C -2.3195,E1 25.065,E2 384.197} C_DIS
LIN {X 33.3389,Y 79.8473,Z 87,A 63.1992,B 24.8965,C -2.3482,E1 25.0581,E2 381.5367} C_DIS
LIN {X 29.3186,Y 81.4097,Z 87,A 65.0265,B 24.8992,C -2.3174,E1 25.0535,E2 379.7864} C_DIS
LIN {X 26.7355,Y 82.2935,Z 87,A 66.6036,B 24.8998,C -2.3115,E1 25.0494,E2 378.2263} C_DIS
LIN {X 24.8714,Y 82.8763,Z 87,A 68.39,B 24.8983,C -2.3283,E1 25.0445,E2 376.4035} C_DIS
LIN {X 19.9576,Y 84.1958,Z 87,A 71.7246,B 24.8983,C -2.3292,E1 25.0355,E2 373.0718} C_DIS
LIN {X 17.5659,Y 84.7258,Z 87,A 74.1757,B 24.8958,C -2.3565,E1 25.0287,E2 370.5589} C_DIS
LIN {X 13.198,Y 85.515,Z 87,A 75.73,B 24.8996,C -2.3134,E1 25.0247,E2 369.1084} C_DIS
LIN {X 9.0796,Y 86.0498,Z 87,A 78.9525,B 24.8982,C -2.3287,E1 25.0156,E2 365.8521} C_DIS
LIN {X 6.6125,Y 86.2749,Z 87,A 81.2199,B 24.8965,C -2.3486,E1 25.0092,E2 363.5386} C_DIS
LIN {X 3.0675,Y 86.4741,Z 87,A 83.1231,B 24.8978,C -2.3343,E1 25.004,E2 361.6699} C_DIS
LIN {X -1.5418,Y 86.5137,Z 87,A 85.9928,B 24.8983,C -2.328,E1 24.996,E2 358.8151} C_DIS
LIN {X -6.6234,Y 86.274,Z 87,A 89.3737,B 24.8983,C -2.3271,E1 24.9866,E2 355.4354} C_DIS
LIN {X -12.5858,Y 85.6082,Z 87,A 93.4405,B 24.8983,C -2.3276,E1 24.9753,E2 351.3645} C_DIS
LIN {X -17.9034,Y 84.6566,Z 87,A 97.0368,B 24.8985,C -2.3254,E1 24.9654,E2 347.7698} C_DIS
LIN {X -23.699,Y 83.2188,Z 87,A 101.1615,B 24.8985,C -2.3266,E1 24.9543,E2 343.6359} C_DIS
LIN {X -29.0944,Y 81.4907,Z 87,A 104.73,B 24.8993,C -2.3166,E1 24.9449,E2 340.0847} C_DIS
LIN {X -32.0797,Y 80.3624,Z 87,A 106.8628,B 24.8995,C -2.3143,E1 24.9393,E2 337.9527} C_DIS
LIN {X -35.0885,Y 79.0952,Z 87,A 109.0401,B 24.8997,C -2.3117,E1 24.9337,E2 335.7766} C_DIS
LIN {X -38.9743,Y 77.2535,Z 87,A 112.2784,B 24.8991,C -2.3188,E1 24.9256,E2 332.5128} C_DIS
LIN {X -42.7057,Y 75.2558,Z 87,A 114.6855,B 24.9006,C -2.3023,E1 24.9198,E2 330.1382} C_DIS
LIN {X -46.7123,Y 72.8352,Z 87,A 118.1703,B 24.9001,C -2.3079,E1 24.9114,E2 326.6291} C_DIS
LIN {X -50.8681,Y 69.9966,Z 87,A 121.9229,B 24.8996,C -2.3136,E1 24.9029,E2 322.8499} C_DIS
LIN {X -54.2234,Y 67.431,Z 87,A 123.9698,B 24.902,C -2.2856,E1 24.8985,E2 320.8622} C_DIS
LIN {X -57.1576,Y 64.9624,Z 87,A 126.4603,B 24.9026,C -2.2785,E1 24.8932,E2 318.3788} C_DIS
LIN {X -60.4223,Y 61.9358,Z 87,A 129.622,B 24.9026,C -2.2778,E1 24.8868,E2 315.2058} C_DIS
LIN {X -63.0632,Y 59.2455,Z 87,A 131.9587,B 24.9036,C -2.2671,E1 24.8823,E2 312.8845} C_DIS
LIN {X -65.8485,Y 56.1336,Z 87,A 135.1469,B 24.9031,C -2.2723,E1 24.8764,E2 309.6695} C_DIS
LIN {X -69.1875,Y 51.9624,Z 87,A 138.3663,B 24.9047,C -2.2537,E1 24.871,E2 306.4791} C_DIS
LIN {X -71.7164,Y 48.4125,Z 87,A 141.1888,B 24.9055,C -2.244,E1 24.8665,E2 303.6659} C_DIS
LIN {X -73.1009,Y 46.2979,Z 87,A 143.0247,B 24.9055,C -2.244,E1 24.8637,E2 301.8209} C_DIS
LIN {X -75.1865,Y 42.8263,Z 87,A 145.6476,B 24.9063,C -2.2346,E1 24.86,E2 299.2066} C_DIS
LIN {X -76.6199,Y 40.2046,Z 87,A 147.7822,B 24.9064,C -2.2333,E1 24.8572,E2 297.0639} C_DIS
LIN {X -78.6714,Y 36.0283,Z 87,A 151.1158,B 24.9066,C -2.2313,E1 24.8532,E2 293.7168} C_DIS
LIN {X -80.5273,Y 31.66,Z 87,A 153.6984,B 24.9087,C -2.2059,E1 24.8505,E2 291.1804} C_DIS
LIN {X -82.635,Y 25.6604,Z 87,A 157.8539,B 24.9099,C -2.1913,E1 24.8468,E2 287.0362} C_DIS
LIN {X -83.8423,Y 21.3891,Z 87,A 161.0978,B 24.9099,C -2.1907,E1 24.8444,E2 283.775} C_DIS
LIN {X -84.6146,Y 18.0969,Z 87,A 163.2735,B 24.9107,C -2.1818,E1 24.843,E2 281.6077} C_DIS
LIN {X -85.142,Y 15.4223,Z 87,A 165.9388,B 24.9092,C -2.2005,E1 24.8417,E2 278.8821} C_DIS
LIN {X -85.8007,Y 11.1912,Z 87,A 167.5109,B 24.9128,C -2.1557,E1 24.8411,E2 277.4074} C_DIS
LIN {X -86.0399,Y 9.1737,Z 87,A 169.536,B 24.9116,C -2.1705,E1 24.8405,E2 275.335} C_DIS
LIN {X -86.3177,Y 6.0239,Z 87,A 171.7247,B 24.912,C -2.1665,E1 24.84,E2 273.1426} C_DIS
LIN {X -86.5115,Y 1.6624,Z 87,A 174.0074,B 24.9141,C -2.1401,E1 24.8398,E2 270.9091} C_DIS
LIN {X -86.4763,Y -2.9953,Z 87,A 177.2432,B 24.9146,C -2.1345,E1 24.8399,E2 267.6674} C_DIS
LIN {X -86.2326,Y -7.1409,Z 87,A -179.7504,B 24.9146,C -2.133,E1 24.8405,E2 264.6465} C_DIS
LIN {X -85.4533,Y -13.5968,Z 87,A -175.4036,B 24.9157,C -2.1205,E1 24.8421,E2 260.3033} C_DIS
LIN {X -84.858,Y -16.9222,Z 87,A -173.1239,B 24.9161,C -2.1148,E1 24.8432,E2 258.0238} C_DIS
LIN {X -83.9096,Y -21.1271,Z 87,A -170.3083,B 24.9169,C -2.105,E1 24.8451,E2 255.2151} C_DIS
LIN {X -83.0753,Y -24.2008,Z 87,A -168.1855,B 24.9174,C -2.099,E1 24.8467,E2 253.0943} C_DIS
LIN {X -81.6923,Y -28.5201,Z 87,A -164.7495,B 24.9171,C -2.1025,E1 24.8497,E2 249.6303} C_DIS
LIN {X -79.7814,Y -33.4955,Z 87,A -161.6116,B 24.9188,C -2.0811,E1 24.8529,E2 246.526} C_DIS
LIN {X -78.511,Y -36.3737,Z 87,A -159.3963,B 24.9189,C -2.079,E1 24.8555,E2 244.3035} C_DIS
LIN {X -76.8886,Y -39.6897,Z 87,A -157.0664,B 24.9197,C -2.069,E1 24.8584,E2 241.9851} C_DIS
LIN {X -73.5351,Y -45.6034,Z 87,A -152.5106,B 24.9205,C -2.0586,E1 24.8648,E2 237.4304} C_DIS
LIN {X -71.6157,Y -48.5613,Z 87,A -149.3172,B 24.919,C -2.0778,E1 24.8699,E2 234.1753} C_DIS
LIN {X -69.0345,Y -52.166,Z 87,A -147.1732,B 24.9214,C -2.0474,E1 24.8734,E2 232.0935} C_DIS
LIN {X -67.4616,Y -54.1856,Z 87,A -145.1916,B 24.9211,C -2.0518,E1 24.8769,E2 230.0922} C_DIS
LIN {X -64.3444,Y -57.8518,Z 87,A -141.9819,B 24.9216,C -2.0453,E1 24.8828,E2 226.8835} C_DIS
LIN {X -61.4047,Y -60.9631,Z 87,A -139.5843,B 24.923,C -2.0263,E1 24.8874,E2 224.5207} C_DIS
LIN {X -59.1133,Y -63.1876,Z 87,A -137.3004,B 24.923,C -2.027,E1 24.892,E2 222.2258} C_DIS
LIN {X -56.9116,Y -65.1772,Z 87,A -135.1333,B 24.9228,C -2.0292,E1 24.8966,E2 220.0449} C_DIS
LIN {X -52.4773,Y -68.799,Z 87,A -131.4932,B 24.9237,C -2.0178,E1 24.9045,E2 216.4185} C_DIS
LIN {X -49.6428,Y -70.8709,Z 87,A -129.2628,B 24.9242,C -2.011,E1 24.9095,E2 214.1963} C_DIS
LIN {X -44.9201,Y -73.9539,Z 87,A -125.5268,B 24.9246,C -2.0053,E1 24.9183,E2 210.4619} C_DIS
LIN {X -40.4542,Y -76.4884,Z 87,A -121.634,B 24.9238,C -2.0158,E1 24.9279,E2 206.5331} C_DIS
LIN {X -36.677,Y -78.3698,Z 87,A -118.3195,B 24.9228,C -2.0286,E1 24.9364,E2 203.1797} C_DIS
LIN {X -32.3309,Y -80.2609,Z 87,A -116.3395,B 24.9258,C -1.9896,E1 24.9413,E2 201.2881} C_DIS
LIN {X -29.8145,Y -81.2288,Z 87,A -114.4848,B 24.9258,C -1.9901,E1 24.9461,E2 199.4283} C_DIS
LIN {X -25.7786,Y -82.5981,Z 87,A -111.1004,B 24.9246,C -2.0053,E1 24.9552,E2 196.0014} C_DIS
LIN {X -21.2452,Y -83.8793,Z 87,A -108.7131,B 24.9265,C -1.9806,E1 24.9615,E2 193.6693} C_DIS
LIN {X -17.518,Y -84.7357,Z 87,A -105.9869,B 24.9261,C -1.9854,E1 24.969,E2 190.9282} C_DIS
LIN {X -12.789,Y -85.5782,Z 87,A -102.6424,B 24.9258,C -1.9895,E1 24.9782,E2 187.5707} C_DIS
LIN {X -9.5561,Y -85.9997,Z 87,A -100.0894,B 24.9249,C -2.0018,E1 24.9854,E2 184.987} C_DIS
LIN {X -4.5364,Y -86.4088,Z 87,A -97.1278,B 24.9258,C -1.9899,E1 24.9936,E2 182.0525} C_DIS
LIN {X -1.0376,Y -86.5227,Z 87,A -94.8048,B 24.9258,C -1.9904,E1 25.0001,E2 179.7281} C_DIS
LIN {X -1.0376,Y -86.5227,Z 87,A -94.8048,B 24.9258,C -1.9904,E1 25.0001,E2 179.7281} C_DIS
Enddeposition()
LIN {X 0.5588,Y -85.6238,Z 87,A -93.0616,B 24.9229,C -2.0281,E1 25.0052,E2 177.8956} C_DIS
Startdeposition()
$VEL.CP = VEL_PRINT
LIN {X -1.4349,Y -85.6216,Z 87,A -96.7178,B 24.9284,C -1.9546,E1 24.9945,E2 181.7263} C_DIS
LIN {X -4.802,Y -85.4988,Z 87,A -98.2674,B 24.9268,C -1.9761,E1 24.9903,E2 183.2251} C_DIS
LIN {X -9.8281,Y -85.0677,Z 87,A -101.7741,B 24.9271,C -1.9723,E1 24.9805,E2 186.7427} C_DIS
LIN {X -14.3789,Y -84.418,Z 87,A -104.9337,B 24.9272,C -1.9705,E1 24.9718,E2 189.9093} C_DIS
LIN {X -19.8131,Y -83.3113,Z 87,A -108.3993,B 24.9265,C -1.9796,E1 24.9624,E2 193.3575} C_DIS
LIN {X -23.3665,Y -82.3838,Z 87,A -112.002,B 24.9289,C -1.9468,E1 24.9525,E2 197.0438} C_DIS
LIN {X -27.861,Y -80.9761,Z 87,A -114.1568,B 24.9266,C -1.9789,E1 24.9469,E2 199.1262} C_DIS
LIN {X -31.7742,Y -79.5219,Z 87,A -117.871,B 24.9284,C -1.9543,E1 24.9371,E2 202.9069} C_DIS
LIN {X -35.772,Y -77.805,Z 87,A -119.9207,B 24.9263,C -1.9828,E1 24.932,E2 204.8937} C_DIS
LIN {X -41.9432,Y -74.6586,Z 87,A -124.3687,B 24.9254,C -1.9942,E1 24.9211,E2 209.3267} C_DIS
LIN {X -44.171,Y -73.3631,Z 87,A -127.5532,B 24.9284,C -1.9544,E1 24.9132,E2 212.6158} C_DIS
LIN {X -48.8506,Y -70.3328,Z 87,A -129.8974,B 24.925,C -2.0003,E1 24.908,E2 214.8586} C_DIS
LIN {X -51.1694,Y -68.6651,Z 87,A -132.9212,B 24.9271,C -1.9716,E1 24.9011,E2 217.9615} C_DIS
LIN {X -54.8099,Y -65.795,Z 87,A -135.188,B 24.9249,C -2.0012,E1 24.8963,E2 220.1666} C_DIS
LIN {X -57.001,Y -63.9062,Z 87,A -136.9998,B 24.9244,C -2.0085,E1 24.8925,E2 221.9681} C_DIS
LIN {X -59.7877,Y -61.3088,Z 87,A -139.6053,B 24.9241,C -2.012,E1 24.8872,E2 224.5758} C_DIS
LIN {X -61.9434,Y -59.1293,Z 87,A -142.3396,B 24.9252,C -1.9971,E1 24.8819,E2 227.3576} C_DIS
LIN {X -64.4886,Y -56.341,Z 87,A -144.8233,B 24.9247,C -2.004,E1 24.8773,E2 229.836} C_DIS
LIN {X -66.8715,Y -53.4934,Z 87,A -146.494,B 24.9225,C -2.0327,E1 24.8745,E2 231.4461} C_DIS
LIN {X -69.7823,Y -49.6341,Z 87,A -150.3675,B 24.9233,C -2.0226,E1 24.868,E2 235.3623} C_DIS
LIN {X -71.7662,Y -46.7221,Z 87,A -152.9584,B 24.9233,C -2.0221,E1 24.864,E2 237.9674} C_DIS
LIN {X -73.677,Y -43.6439,Z 87,A -155.2453,B 24.9226,C -2.0323,E1 24.8608,E2 240.2418} C_DIS
LIN {X -75.2586,Y -40.8562,Z 87,A -156.4148,B 24.92,C -2.0652,E1 24.8593,E2 241.339} C_DIS
LIN {X -76.1223,Y -39.2246,Z 87,A -158.1473,B 24.9208,C -2.0547,E1 24.857,E2 243.1059} C_DIS
LIN {X -77.9447,Y -35.4656,Z 87,A -160.9585,B 24.9203,C -2.062,E1 24.8536,E2 245.9148} C_DIS
LIN {X -79.1477,Y -32.6945,Z 87,A -163.6401,B 24.9212,C -2.0497,E1 24.8507,E2 248.6408} C_DIS
LIN {X -80.4586,Y -29.3174,Z 87,A -165.1573,B 24.9187,C -2.0817,E1 24.8493,E2 250.0902} C_DIS
LIN {X -81.9389,Y -24.8862,Z 87,A -168.3653,B 24.9182,C -2.0886,E1 24.8465,E2 253.3} C_DIS
LIN {X -82.9806,Y -21.1503,Z 87,A -171.6146,B 24.919,C -2.0786,E1 24.8441,E2 256.5921} C_DIS
LIN {X -83.7668,Y -17.7888,Z 87,A -173.5182,B 24.9176,C -2.0967,E1 24.843,E2 258.4637} C_DIS
LIN {X -84.2894,Y -15.1128,Z 87,A -175.3672,B 24.9172,C -2.1017,E1 24.8421,E2 260.3117} C_DIS
LIN {X -85.1184,Y -9.3898,Z 87,A -179.3154,B 24.9164,C -2.1116,E1 24.8406,E2 264.2598} C_DIS
LIN {X -85.4005,Y -6.3314,Z 87,A 178.5602,B 24.916,C -2.1163,E1 24.8401,E2 266.3859} C_DIS
LIN {X -85.5834,Y -2.9445,Z 87,A 175.8878,B 24.9163,C -2.1126,E1 24.8398,E2 269.0832} C_DIS
LIN {X -85.6342,Y 0.3189,Z 87,A 174.4934,B 24.914,C -2.141,E1 24.8398,E2 270.4182} C_DIS
LIN {X -85.5422,Y 3.9618,Z 87,A 171.6852,B 24.9142,C -2.1387,E1 24.84,E2 273.2488} C_DIS
LIN {X -85.0154,Y 10.2748,Z 87,A 167.7274,B 24.9125,C -2.1599,E1 24.8411,E2 277.1797} C_DIS
LIN {X -84.2296,Y 15.4451,Z 87,A 164.105,B 24.9119,C -2.1676,E1 24.8426,E2 280.8051} C_DIS
LIN {X -83.8376,Y 17.447,Z 87,A 162.5243,B 24.9119,C -2.166,E1 24.8435,E2 282.3989} C_DIS
LIN {X -83.0894,Y 20.7228,Z 87,A 159.3748,B 24.9134,C -2.1488,E1 24.8457,E2 285.608} C_DIS
LIN {X -81.8708,Y 25.1064,Z 87,A 157.5806,B 24.9099,C -2.1921,E1 24.847,E2 287.3091} C_DIS
LIN {X -80.0334,Y 30.4591,Z 87,A 153.4231,B 24.9097,C -2.1936,E1 24.8509,E2 291.4867} C_DIS
LIN {X -77.7621,Y 35.8642,Z 87,A 149.4909,B 24.9088,C -2.2051,E1 24.8552,E2 295.4131} C_DIS
LIN {X -75.6972,Y 40.038,Z 87,A 146.61,B 24.9075,C -2.2208,E1 24.8588,E2 298.2723} C_DIS
LIN {X -74.5559,Y 42.1272,Z 87,A 144.4481,B 24.9084,C -2.2097,E1 24.8618,E2 300.4719} C_DIS
LIN {X -72.4067,Y 45.7223,Z 87,A 141.8668,B 24.9072,C -2.2237,E1 24.8655,E2 303.033} C_DIS
LIN {X -70.5567,Y 48.5285,Z 87,A 139.1268,B 24.9078,C -2.2164,E1 24.8699,E2 305.804} C_DIS
LIN {X -68.6523,Y 51.1864,Z 87,A 137.3256,B 24.9065,C -2.2329,E1 24.8728,E2 307.5746} C_DIS
LIN {X -65.8454,Y 54.7491,Z 87,A 134.4703,B 24.9054,C -2.2458,E1 24.8778,E2 310.4125} C_DIS
LIN {X -62.9839,Y 58.0176,Z 87,A 131.4263,B 24.9051,C -2.2493,E1 24.8834,E2 313.4617} C_DIS
LIN {X -60.3791,Y 60.7235,Z 87,A 128.6874,B 24.9051,C -2.2491,E1 24.8888,E2 316.2128} C_DIS
LIN {X -57.2536,Y 63.6801,Z 87,A 125.166,B 24.9061,C -2.2379,E1 24.8962,E2 319.7751} C_DIS
LIN {X -53.8691,Y 66.5674,Z 87,A 122.5112,B 24.9048,C -2.2532,E1 24.9019,E2 322.4032} C_DIS
LIN {X -51.1739,Y 68.6616,Z 87,A 120.9825,B 24.9025,C -2.2792,E1 24.9052,E2 323.8756} C_DIS
LIN {X -49.0907,Y 70.166,Z 87,A 119.0401,B 24.9028,C -2.2763,E1 24.9096,E2 325.8315} C_DIS
LIN {X -45.7217,Y 72.407,Z 87,A 115.7058,B 24.9039,C -2.2638,E1 24.9175,E2 329.2065} C_DIS
LIN {X -42.6821,Y 74.2383,Z 87,A 113.9766,B 24.9019,C -2.2863,E1 24.9216,E2 330.8873} C_DIS
LIN {X -37.9345,Y 76.7729,Z 87,A 109.9144,B 24.9026,C -2.279,E1 24.9317,E2 334.9779} C_DIS
LIN {X -34.3762,Y 78.4308,Z 87,A 107.7161,B 24.9012,C -2.2952,E1 24.9372,E2 337.143} C_DIS
LIN {X -31.3268,Y 79.6977,Z 87,A 105.0433,B 24.9021,C -2.2849,E1 24.9442,E2 339.8463} C_DIS
LIN {X -26.1967,Y 81.5283,Z 87,A 101.3302,B 24.9018,C -2.2873,E1 24.9541,E2 343.5606} C_DIS
LIN {X -19.7417,Y 83.3282,Z 87,A 97.0145,B 24.901,C -2.2966,E1 24.9657,E2 347.8604} C_DIS
LIN {X -15.6888,Y 84.1856,Z 87,A 94.4975,B 24.9002,C -2.3064,E1 24.9725,E2 350.3571} C_DIS
LIN {X -12.3581,Y 84.7376,Z 87,A 91.6241,B 24.9016,C -2.2898,E1 24.9806,E2 353.2724} C_DIS
LIN {X -8.6638,Y 85.1944,Z 87,A 89.9587,B 24.8994,C -2.3156,E1 24.985,E2 354.8774} C_DIS
LIN {X -3.5392,Y 85.5604,Z 87,A 86.8625,B 24.8984,C -2.3273,E1 24.9936,E2 357.9471} C_DIS
LIN {X 0.0737,Y 85.6344,Z 87,A 84.0799,B 24.8993,C -2.3168,E1 25.0014,E2 360.7547} C_DIS
LIN {X 2.2542,Y 85.6046,Z 87,A 81.4723,B 24.9023,C -2.2824,E1 25.0089,E2 363.4434} C_DIS
LIN {X 7.0465,Y 85.3433,Z 87,A 79.1714,B 24.8999,C -2.3097,E1 25.0151,E2 365.6784} C_DIS
LIN {X 12.5704,Y 84.7074,Z 87,A 75.7209,B 24.8993,C -2.3172,E1 25.0247,E2 369.1084} C_DIS
LIN {X 16.6754,Y 83.9956,Z 87,A 72.9661,B 24.8993,C -2.3172,E1 25.0322,E2 371.8604} C_DIS
LIN {X 20.4698,Y 83.1511,Z 87,A 69.1441,B 24.9026,C -2.2782,E1 25.0428,E2 375.7693} C_DIS
LIN {X 25.1641,Y 81.8529,Z 87,A 66.9866,B 24.8999,C -2.3099,E1 25.0484,E2 377.8479} C_DIS
LIN {X 28.7722,Y 80.6564,Z 87,A 63.3206,B 24.9031,C -2.2727,E1 25.0583,E2 381.5945} C_DIS
LIN {X 33.3673,Y 78.8652,Z 87,A 61.3729,B 24.8997,C -2.3117,E1 25.063,E2 383.4455} C_DIS
LIN {X 38.3932,Y 76.5443,Z 87,A 57.4088,B 24.9008,C -2.299,E1 25.0731,E2 387.4295} C_DIS
LIN {X 41.2255,Y 75.0583,Z 87,A 54.1904,B 24.904,C -2.262,E1 25.0812,E2 390.7261} C_DIS
LIN {X 45.506,Y 72.5419,Z 87,A 51.9273,B 24.9016,C -2.2906,E1 25.0864,E2 392.9144} C_DIS
LIN {X 48.241,Y 70.7529,Z 87,A 49.7343,B 24.9019,C -2.2869,E1 25.0915,E2 395.1088} C_DIS
LIN {X 51.8189,Y 68.1772,Z 87,A 46.4548,B 24.9032,C -2.2711,E1 25.0989,E2 398.4139} C_DIS
LIN {X 54.7444,Y 65.8494,Z 87,A 44.3751,B 24.9025,C -2.2801,E1 25.1033,E2 400.4644} C_DIS
LIN {X 58.5022,Y 62.535,Z 87,A 41.3468,B 24.9021,C -2.2841,E1 25.1096,E2 403.4713} C_DIS
LIN {X 60.142,Y 60.9593,Z 87,A 39.528,B 24.9032,C -2.2712,E1 25.1133,E2 405.3131} C_DIS
LIN {X 64.8311,Y 55.9488,Z 87,A 34.9324,B 24.9041,C -2.2608,E1 25.122,E2 409.9129} C_DIS
LIN {X 66.8994,Y 53.4581,Z 87,A 32.2799,B 24.9059,C -2.2398,E1 25.1267,E2 412.6029} C_DIS
LIN {X 69.9886,Y 49.345,Z 87,A 29.4956,B 24.9048,C -2.253,E1 25.1312,E2 415.3425} C_DIS
LIN {X 71.5558,Y 47.0411,Z 87,A 27.245,B 24.9063,C -2.2355,E1 25.1348,E2 417.6234} C_DIS
LIN {X 73.6212,Y 43.7384,Z 87,A 24.8775,B 24.9062,C -2.2366,E1 25.1382,E2 419.9762} C_DIS
LIN {X 75.93,Y 39.5961,Z 87,A 21.298,B 24.908,C -2.2144,E1 25.143,E2 423.5892} C_DIS
LIN {X 77.9152,Y 35.5312,Z 87,A 17.4123,B 24.9111,C -2.1775,E1 25.1476,E2 427.5411} C_DIS
LIN {X 80.1366,Y 30.1867,Z 87,A 15.0321,B 24.9079,C -2.216,E1 25.1499,E2 429.8172} C_DIS
LIN {X 81.1188,Y 27.438,Z 87,A 12.9709,B 24.9087,C -2.2066,E1 25.1518,E2 431.8891} C_DIS
LIN {X 82.7118,Y 22.1783,Z 87,A 9.3067,B 24.9095,C -2.1959,E1 25.1547,E2 435.5574} C_DIS
LIN {X 83.4537,Y 19.1984,Z 87,A 6.4596,B 24.9123,C -2.163,E1 25.1565,E2 438.4658} C_DIS
LIN {X 84.277,Y 15.1817,Z 87,A 4.4232,B 24.911,C -2.1782,E1 25.1576,E2 440.4542} C_DIS
LIN {X 85.067,Y 9.8342,Z 87,A 0.871,B 24.9118,C -2.1691,E1 25.1589,E2 444.0071} C_DIS
LIN {X 85.4501,Y 5.6001,Z 87,A -1.9291,B 24.9124,C -2.1616,E1 25.1595,E2 446.8084} C_DIS
LIN {X 85.6112,Y 1.9558,Z 87,A -4.5152,B 24.9134,C -2.1488,E1 25.1598,E2 449.4091} C_DIS
LIN {X 85.6179,Y -1.6313,Z 87,A -7.2567,B 24.9149,C -2.1296,E1 25.1597,E2 452.1797} C_DIS
LIN {X 85.4885,Y -4.9823,Z 87,A -8.6976,B 24.9133,C -2.1497,E1 25.1595,E2 453.5647} C_DIS
LIN {X 85.1356,Y -9.2261,Z 87,A -11.6126,B 24.9142,C -2.1383,E1 25.1588,E2 456.4893} C_DIS
LIN {X 84.7819,Y -12.0469,Z 87,A -14.691,B 24.9179,C -2.0924,E1 25.1575,E2 459.6578} C_DIS
LIN {X 83.9459,Y -16.9197,Z 87,A -16.6418,B 24.9151,C -2.1278,E1 25.1566,E2 461.5136} C_DIS
LIN {X 82.9766,Y -21.1658,Z 87,A -19.4841,B 24.9156,C -2.121,E1 25.1548,E2 464.3555} C_DIS
LIN {X 82.3453,Y -23.5027,Z 87,A -21.7781,B 24.9179,C -2.093,E1 25.153,E2 466.7025} C_DIS
LIN {X 81.0875,Y -27.5309,Z 87,A -25.0114,B 24.9196,C -2.0704,E1 25.1501,E2 469.9709} C_DIS
LIN {X 79.6987,Y -31.3242,Z 87,A -26.4326,B 24.9169,C -2.1055,E1 25.1488,E2 471.3012} C_DIS
LIN {X 78.889,Y -33.3109,Z 87,A -28.633,B 24.9192,C -2.0751,E1 25.1464,E2 473.5613} C_DIS
LIN {X 77.0967,Y -37.2723,Z 87,A -31.2053,B 24.919,C -2.0778,E1 25.1434,E2 476.1133} C_DIS
LIN {X 75.7056,Y -40.022,Z 87,A -33.9617,B 24.9213,C -2.0484,E1 25.1397,E2 478.9247} C_DIS
LIN {X 73.8818,Y -43.2975,Z 87,A -35.8259,B 24.9202,C -2.0628,E1 25.1372,E2 480.7452} C_DIS
LIN {X 71.9967,Y -46.3636,Z 87,A -38.1863,B 24.9206,C -2.0576,E1 25.1337,E2 483.106} C_DIS
LIN {X 70.3172,Y -48.8731,Z 87,A -40.4832,B 24.9218,C -2.0427,E1 25.13,E2 485.4267} C_DIS
LIN {X 67.6142,Y -52.5504,Z 87,A -43.1986,B 24.9215,C -2.0458,E1 25.1255,E2 488.1217} C_DIS
LIN {X 65.696,Y -54.929,Z 87,A -45.4633,B 24.9225,C -2.0331,E1 25.1214,E2 490.406} C_DIS
LIN {X 63.6973,Y -57.2344,Z 87,A -47.4718,B 24.9228,C -2.029,E1 25.1177,E2 492.4152} C_DIS
LIN {X 60.4426,Y -60.6624,Z 87,A -50.7488,B 24.9237,C -2.0175,E1 25.1113,E2 495.7054} C_DIS
LIN {X 56.5433,Y -64.3119,Z 87,A -53.677,B 24.9227,C -2.0306,E1 25.1053,E2 498.5906} C_DIS
LIN {X 54.6642,Y -65.9161,Z 87,A -56.0635,B 24.9248,C -2.0026,E1 25.1001,E2 501.0342} C_DIS
LIN {X 50.7317,Y -68.9885,Z 87,A -59.1715,B 24.9248,C -2.0032,E1 25.0932,E2 504.1296} C_DIS
LIN {X 47.4155,Y -71.309,Z 87,A -61.9306,B 24.9253,C -1.9961,E1 25.0868,E2 506.8961} C_DIS
LIN {X 43.4949,Y -73.7651,Z 87,A -65.2491,B 24.9263,C -1.9832,E1 25.0789,E2 510.2349} C_DIS
LIN {X 40.6851,Y -75.3515,Z 87,A -66.9467,B 24.9254,C -1.9944,E1 25.0748,E2 511.901} C_DIS
LIN {X 36.2239,Y -77.5946,Z 87,A -70.097,B 24.9254,C -1.9952,E1 25.0669,E2 515.041} C_DIS
LIN {X 34.4712,Y -78.389,Z 87,A -72.2086,B 24.9275,C -1.9667,E1 25.0614,E2 517.215} C_DIS
LIN {X 30.8618,Y -79.8804,Z 87,A -73.9141,B 24.9256,C -1.9922,E1 25.0571,E2 518.8562} C_DIS
LIN {X 26.437,Y -81.4505,Z 87,A -77.2251,B 24.9263,C -1.9828,E1 25.0483,E2 522.183} C_DIS
LIN {X 24.0303,Y -82.1934,Z 87,A -78.9399,B 24.9265,C -1.9799,E1 25.0437,E2 523.9015} C_DIS
LIN {X 20.9018,Y -83.0445,Z 87,A -81.985,B 24.9287,C -1.95,E1 25.0353,E2 527.013} C_DIS
LIN {X 16.5536,Y -84.0191,Z 87,A -84.0832,B 24.9268,C -1.9752,E1 25.0297,E2 529.0487} C_DIS
LIN {X 11.1777,Y -84.901,Z 87,A -87.6638,B 24.9268,C -1.9747,E1 25.0199,E2 532.6273} C_DIS
LIN {X 5.4843,Y -85.4582,Z 87,A -91.2148,B 24.9264,C -1.9813,E1 25.01,E2 536.1604} C_DIS
LIN {X 0.5588,Y -85.6238,Z 87,A -93.0577,B 24.923,C -2.0265,E1 25.0053,E2 537.8955} C_DIS
Enddeposition()
LIN {X 0.5588,Y -85.6238,Z 87,A -93.0577,B 24.923,C -2.0265,E1 25.0053,E2 537.8955} C_DIS
Startdeposition()
$VEL.CP = VEL_PRINT
LIN {X 3.2953,Y -84.6752,Z 87,A -91.7802,B 24.9232,C -2.0239,E1 25.0087,E2 536.6245} C_DIS
LIN {X 7.1908,Y -84.4338,Z 87,A -89.1325,B 24.9231,C -2.0254,E1 25.0161,E2 533.9745} C_DIS
LIN {X 11.1329,Y -84.0053,Z 87,A -86.7641,B 24.9237,C -2.0171,E1 25.0226,E2 531.6276} C_DIS
LIN {X 14.0687,Y -83.5635,Z 87,A -84.4236,B 24.9228,C -2.0293,E1 25.0291,E2 529.2607} C_DIS
LIN {X 16.9072,Y -83.0358,Z 87,A -82.1895,B 24.922,C -2.04,E1 25.0353,E2 527.0039} C_DIS
LIN {X 20.1754,Y -82.3027,Z 87,A -80.5572,B 24.9234,C -2.0218,E1 25.0396,E2 525.417} C_DIS
LIN {X 23.0765,Y -81.5368,Z 87,A -78.5364,B 24.9232,C -2.0237,E1 25.0451,E2 523.3949} C_DIS
LIN {X 26.3569,Y -80.5368,Z 87,A -75.6393,B 24.9216,C -2.0452,E1 25.0529,E2 520.4523} C_DIS
LIN {X 29.4042,Y -79.4753,Z 87,A -74.045,B 24.9228,C -2.029,E1 25.057,E2 518.8999} C_DIS
LIN {X 34.5411,Y -77.3807,Z 87,A -70.533,B 24.923,C -2.0265,E1 25.066,E2 515.4018} C_DIS
LIN {X 38.7945,Y -75.3382,Z 87,A -67.065,B 24.9219,C -2.0407,E1 25.0748,E2 511.9094} C_DIS
LIN {X 41.0525,Y -74.132,Z 87,A -65.05,B 24.921,C -2.0531,E1 25.0797,E2 509.871} C_DIS
LIN {X 47.0981,Y -70.4471,Z 87,A -60.7226,B 24.9214,C -2.0468,E1 25.0899,E2 505.5721} C_DIS
LIN {X 48.6928,Y -69.3536,Z 87,A -59.0972,B 24.9204,C -2.0601,E1 25.0937,E2 503.9211} C_DIS
LIN {X 51.7256,Y -67.1211,Z 87,A -56.6415,B 24.9202,C -2.0624,E1 25.0992,E2 501.4687} C_DIS
LIN {X 54.8996,Y -64.5509,Z 87,A -54.0654,B 24.9202,C -2.0624,E1 25.1047,E2 498.9027} C_DIS
LIN {X 57.0362,Y -62.6712,Z 87,A -51.9399,B 24.9194,C -2.0735,E1 25.1091,E2 496.7592} C_DIS
LIN {X 59.818,Y -60.0228,Z 87,A -49.385,B 24.919,C -2.0783,E1 25.1142,E2 494.2037} C_DIS
LIN {X 62.5166,Y -57.2054,Z 87,A -46.9078,B 24.919,C -2.0795,E1 25.119,E2 491.7346} C_DIS
LIN {X 64.3306,Y -55.1582,Z 87,A -44.8206,B 24.9179,C -2.0922,E1 25.1228,E2 489.6266} C_DIS
LIN {X 66.9627,Y -51.9312,Z 87,A -42.2643,B 24.918,C -2.0909,E1 25.1272,E2 487.0855} C_DIS
LIN {X 68.6847,Y -49.6309,Z 87,A -39.9732,B 24.9167,C -2.108,E1 25.1311,E2 484.7651} C_DIS
LIN {X 70.663,Y -46.7712,Z 87,A -37.5474,B 24.9159,C -2.1171,E1 25.1349,E2 482.3298} C_DIS
LIN {X 73.386,Y -42.3711,Z 87,A -34.1057,B 24.9153,C -2.1251,E1 25.1398,E2 478.8867} C_DIS
LIN {X 75.5093,Y -38.4596,Z 87,A -31.4878,B 24.9157,C -2.1205,E1 25.1431,E2 476.2935} C_DIS
LIN {X 76.6847,Y -36.0604,Z 87,A -29.6554,B 24.9152,C -2.1268,E1 25.1453,E2 474.4561} C_DIS
LIN {X 78.3131,Y -32.3737,Z 87,A -27.0096,B 24.9147,C -2.1323,E1 25.1483,E2 471.8118} C_DIS
LIN {X 80.1716,Y -27.4468,Z 87,A -23.7175,B 24.9146,C -2.1341,E1 25.1515,E2 468.5338} C_DIS
LIN {X 81.3554,Y -23.7118,Z 87,A -20.6975,B 24.9129,C -2.155,E1 25.1539,E2 465.4817} C_DIS
LIN {X 82.2538,Y -20.376,Z 87,A -18.0274,B 24.9114,C -2.1739,E1 25.1558,E2 462.7824} C_DIS
LIN {X 83.0294,Y -16.9382,Z 87,A -15.4858,B 24.9103,C -2.1869,E1 25.1572,E2 460.2249} C_DIS
LIN {X 83.6845,Y -13.3353,Z 87,A -13.63,B 24.9114,C -2.1734,E1 25.1581,E2 458.4118} C_DIS
LIN {X 84.1445,Y -10.0258,Z 87,A -11.4282,B 24.911,C -2.1787,E1 25.1588,E2 456.2106} C_DIS
LIN {X 84.3647,Y -7.9625,Z 87,A -9.7118,B 24.9097,C -2.194,E1 25.1593,E2 454.4683} C_DIS
LIN {X 84.7348,Y -1.0284,Z 87,A -5.619,B 24.9102,C -2.1883,E1 25.1598,E2 450.4132} C_DIS
LIN {X 84.6723,Y 3.3794,Z 87,A -2.7531,B 24.9097,C -2.1939,E1 25.1597,E2 447.5512} C_DIS
LIN {X 84.2544,Y 9.0572,Z 87,A 1.0635,B 24.9088,C -2.2049,E1 25.1588,E2 443.7313} C_DIS
LIN {X 83.4407,Y 14.7808,Z 87,A 4.9455,B 24.9079,C -2.2161,E1 25.1573,E2 439.8456} C_DIS
LIN {X 82.7053,Y 18.4601,Z 87,A 7.8319,B 24.9062,C -2.2358,E1 25.1556,E2 436.9295} C_DIS
LIN {X 81.9585,Y 21.5356,Z 87,A 9.7792,B 24.9062,C -2.2358,E1 25.1543,E2 434.9935} C_DIS
LIN {X 80.7931,Y 25.5634,Z 87,A 12.8189,B 24.9049,C -2.2512,E1 25.1519,E2 431.9347} C_DIS
LIN {X 79.7891,Y 28.5437,Z 87,A 14.9089,B 24.9045,C -2.2562,E1 25.1499,E2 429.8446} C_DIS
LIN {X 77.7988,Y 33.5877,Z 87,A 18.5397,B 24.9037,C -2.2656,E1 25.1461,E2 426.2117} C_DIS
LIN {X 76.4555,Y 36.5428,Z 87,A 22.0256,B 24.8994,C -2.3157,E1 25.1418,E2 422.6262} C_DIS
LIN {X 73.7543,Y 41.7289,Z 87,A 24.6901,B 24.9023,C -2.2825,E1 25.1383,E2 420.0541} C_DIS
LIN {X 72.159,Y 44.4308,Z 87,A 26.8787,B 24.9016,C -2.2903,E1 25.1351,E2 417.8582} C_DIS
LIN {X 70.0783,Y 47.6428,Z 87,A 29.1884,B 24.9018,C -2.2877,E1 25.1316,E2 415.5662} C_DIS
LIN {X 68.631,Y 49.7067,Z 87,A 31.884,B 24.8986,C -2.3251,E1 25.1271,E2 412.7953} C_DIS
LIN {X 65.9938,Y 53.157,Z 87,A 34.0178,B 24.9003,C -2.3052,E1 25.1234,E2 410.7185} C_DIS
LIN {X 64.1667,Y 55.3506,Z 87,A 36.6576,B 24.8979,C -2.3332,E1 25.1185,E2 408.0243} C_DIS
LIN {X 61.3788,Y 58.4267,Z 87,A 38.7531,B 24.8994,C -2.3157,E1 25.1146,E2 405.9794} C_DIS
LIN {X 58.936,Y 60.8881,Z 87,A 40.9678,B 24.8994,C -2.3163,E1 25.1102,E2 403.7725} C_DIS
LIN {X 56.9503,Y 62.7507,Z 87,A 42.6262,B 24.8995,C -2.314,E1 25.1068,E2 402.1263} C_DIS
LIN {X 54.6228,Y 64.7867,Z 87,A 44.9798,B 24.8984,C -2.3267,E1 25.1018,E2 399.752} C_DIS
LIN {X 51.6895,Y 67.1489,Z 87,A 47.1629,B 24.8991,C -2.3195,E1 25.0971,E2 397.594} C_DIS
LIN {X 48.2353,Y 69.6718,Z 87,A 50.3703,B 24.8977,C -2.3346,E1 25.0898,E2 394.362} C_DIS
LIN {X 45.9019,Y 71.2307,Z 87,A 52.6473,B 24.8964,C -2.3499,E1 25.0844,E2 392.0563} C_DIS
LIN {X 40.464,Y 74.4544,Z 87,A 56.4157,B 24.8973,C -2.3396,E1 25.0753,E2 388.3236} C_DIS
LIN {X 34.6005,Y 77.354,Z 87,A 60.9068,B 24.8966,C -2.3471,E1 25.064,E2 383.8266} C_DIS
LIN {X 31.4842,Y 78.6746,Z 87,A 63.6816,B 24.8951,C -2.3649,E1 25.0567,E2 381.016} C_DIS
LIN {X 28.4517,Y 79.8214,Z 87,A 65.3889,B 24.8962,C -2.3515,E1 25.0524,E2 379.344} C_DIS
LIN {X 25.1997,Y 80.9059,Z 87,A 67.368,B 24.897,C -2.3427,E1 25.0472,E2 377.3894} C_DIS
LIN {X 20.8203,Y 82.1424,Z 87,A 70.7957,B 24.8959,C -2.3557,E1 25.0379,E2 373.9365} C_DIS
LIN {X 17.4595,Y 82.9224,Z 87,A 73.1298,B 24.8958,C -2.3568,E1 25.0315,E2 371.6027} C_DIS
LIN {X 13.1736,Y 83.7095,Z 87,A 75.9179,B 24.8961,C -2.353,E1 25.0239,E2 368.8267} C_DIS
LIN {X 7.4604,Y 84.4111,Z 87,A 79.9165,B 24.8958,C -2.3569,E1 25.0128,E2 364.8218} C_DIS
LIN {X 3.3792,Y 84.6716,Z 87,A 82.7607,B 24.8956,C -2.3592,E1 25.0048,E2 361.973} C_DIS
LIN {X -0.2523,Y 84.739,Z 87,A 85.376,B 24.8952,C -2.3637,E1 24.9975,E2 359.3473} C_DIS
LIN {X -4.2156,Y 84.6358,Z 87,A 87.6475,B 24.8963,C -2.3504,E1 24.9912,E2 357.107} C_DIS
LIN {X -7.2608,Y 84.4294,Z 87,A 90.0314,B 24.8956,C -2.3591,E1 24.9845,E2 354.7013} C_DIS
LIN {X -12.1304,Y 83.867,Z 87,A 93.0994,B 24.8964,C -2.3498,E1 24.9761,E2 351.6533} C_DIS
LIN {X -15.0881,Y 83.3855,Z 87,A 95.2821,B 24.8961,C -2.353,E1 24.9701,E2 349.4609} C_DIS
LIN {X -19.9488,Y 82.358,Z 87,A 98.9222,B 24.8956,C -2.3583,E1 24.9601,E2 345.8033} C_DIS
LIN {X -26.4161,Y 80.5173,Z 87,A 103.1612,B 24.8969,C -2.3442,E1 24.9488,E2 341.5909} C_DIS
LIN {X -30.267,Y 79.1502,Z 87,A 106.3862,B 24.896,C -2.3542,E1 24.9403,E2 338.3354} C_DIS
LIN {X -34.9739,Y 77.1857,Z 87,A 109.6037,B 24.897,C -2.3424,E1 24.9321,E2 335.1384} C_DIS
LIN {X -39.6657,Y 74.8829,Z 87,A 113.0678,B 24.8977,C -2.3347,E1 24.9235,E2 331.6834} C_DIS
LIN {X -42.4977,Y 73.3132,Z 87,A 115.4981,B 24.8975,C -2.3378,E1 24.9176,E2 329.2385} C_DIS
LIN {X -46.3868,Y 70.9164,Z 87,A 118.1972,B 24.8989,C -2.3208,E1 24.9113,E2 326.5714} C_DIS
LIN {X -48.8526,Y 69.2416,Z 87,A 120.2741,B 24.8991,C -2.3185,E1 24.9065,E2 324.4927} C_DIS
LIN {X -51.4842,Y 67.3071,Z 87,A 122.7911,B 24.8988,C -2.3228,E1 24.9009,E2 321.9567} C_DIS
LIN {X -56.1078,Y 63.5053,Z 87,A 126.628,B 24.9001,C -2.3078,E1 24.8927,E2 318.1406} C_DIS
LIN {X -58.648,Y 61.1657,Z 87,A 128.5203,B 24.9016,C -2.2899,E1 24.889,E2 316.2832} C_DIS
LIN {X -61.4143,Y 58.3886,Z 87,A 132.1424,B 24.8998,C -2.3108,E1 24.8818,E2 312.5956} C_DIS
LIN {X -63.7213,Y 55.8606,Z 87,A 133.8667,B 24.9017,C -2.2884,E1 24.8787,E2 310.9171} C_DIS
LIN {X -66.0994,Y 53.0265,Z 87,A 136.9351,B 24.9009,C -2.2978,E1 24.8732,E2 307.812} C_DIS
LIN {X -68.1163,Y 50.4094,Z 87,A 139.0324,B 24.9018,C -2.288,E1 24.8697,E2 305.7281} C_DIS
LIN {X -70.511,Y 47.0017,Z 87,A 141.5327,B 24.9032,C -2.2714,E1 24.8658,E2 303.2549} C_DIS
LIN {X -72.3206,Y 44.165,Z 87,A 143.4005,B 24.9047,C -2.2538,E1 24.8631,E2 301.4196} C_DIS
LIN {X -73.9235,Y 41.426,Z 87,A 145.9049,B 24.9044,C -2.2575,E1 24.8596,E2 298.8933} C_DIS
LIN {X -76.5328,Y 36.3819,Z 87,A 149.5733,B 24.9057,C -2.2415,E1 24.855,E2 295.2435} C_DIS
LIN {X -77.6776,Y 33.8668,Z 87,A 151.7405,B 24.9055,C -2.2441,E1 24.8525,E2 293.0582} C_DIS
LIN {X -79.184,Y 30.1779,Z 87,A 155.204,B 24.9044,C -2.2572,E1 24.849,E2 289.5438} C_DIS
LIN {X -80.5714,Y 26.2488,Z 87,A 156.925,B 24.9077,C -2.2182,E1 24.8475,E2 287.9061} C_DIS
LIN {X -82.3326,Y 20.053,Z 87,A 161.6048,B 24.9081,C -2.2134,E1 24.844,E2 283.2107} C_DIS
LIN {X -82.8418,Y 17.8346,Z 87,A 163.5048,B 24.9077,C -2.2185,E1 24.8429,E2 281.2875} C_DIS
LIN {X -83.5111,Y 14.3821,Z 87,A 165.7916,B 24.9085,C -2.2084,E1 24.8418,E2 279.0112} C_DIS
LIN {X -84.1488,Y 9.9886,Z 87,A 169.4364,B 24.9078,C -2.2166,E1 24.8405,E2 275.3249} C_DIS
LIN {X -84.5474,Y 5.7021,Z 87,A 171.4346,B 24.9107,C -2.1821,E1 24.8401,E2 273.3972} C_DIS
LIN {X -84.7019,Y 2.5245,Z 87,A 173.6694,B 24.9111,C -2.1775,E1 24.8398,E2 271.1599} C_DIS
LIN {X -84.7406,Y -0.2627,Z 87,A 175.9222,B 24.9107,C -2.1816,E1 24.8398,E2 268.8837} C_DIS
LIN {X -84.5906,Y -5.0339,Z 87,A 178.8012,B 24.9124,C -2.1617,E1 24.8402,E2 266.0348} C_DIS
LIN {X -84.3581,Y -8.0346,Z 87,A -179.159,B 24.9129,C -2.1554,E1 24.8407,E2 263.9978} C_DIS
LIN {X -84.1106,Y -10.3152,Z 87,A -177.1221,B 24.9122,C -2.164,E1 24.8414,E2 261.9284} C_DIS
LIN {X -83.4038,Y -14.9864,Z 87,A -174.4155,B 24.9141,C -2.1405,E1 24.8426,E2 259.2616} C_DIS
LIN {X -82.8141,Y -17.9616,Z 87,A -172.3049,B 24.9144,C -2.1359,E1 24.8438,E2 257.1497} C_DIS
LIN {X -81.8716,Y -21.8606,Z 87,A -169.5463,B 24.915,C -2.1289,E1 24.8456,E2 254.3916} C_DIS
LIN {X -81.2391,Y -24.1035,Z 87,A -167.4323,B 24.9142,C -2.1392,E1 24.8474,E2 252.2409} C_DIS
LIN {X -80.2424,Y -27.2392,Z 87,A -165.7909,B 24.916,C -2.1163,E1 24.8488,E2 250.6447} C_DIS
LIN {X -78.5558,Y -31.7774,Z 87,A -162.4415,B 24.9166,C -2.1089,E1 24.8521,E2 247.2941} C_DIS
LIN {X -77.2508,Y -34.8295,Z 87,A -160.3349,B 24.9174,C -2.0987,E1 24.8545,E2 245.2003} C_DIS
LIN {X -75.9258,Y -37.6304,Z 87,A -158.052,B 24.9174,C -2.0981,E1 24.8572,E2 242.9064} C_DIS
LIN {X -74.5345,Y -40.3162,Z 87,A -155.5529,B 24.9169,C -2.1054,E1 24.8606,E2 240.3768} C_DIS
LIN {X -71.5117,Y -45.4641,Z 87,A -151.9534,B 24.9187,C -2.0824,E1 24.8657,E2 236.8136} C_DIS
LIN {X -69.9786,Y -47.79,Z 87,A -149.005,B 24.9167,C -2.1081,E1 24.8705,E2 233.7892} C_DIS
LIN {X -67.1102,Y -51.7397,Z 87,A -146.8378,B 24.9198,C -2.0676,E1 24.874,E2 231.7082} C_DIS
LIN {X -64.6357,Y -54.8001,Z 87,A -143.9383,B 24.9198,C -2.0683,E1 24.8792,E2 228.7938} C_DIS
LIN {X -61.3069,Y -58.5014,Z 87,A -140.6117,B 24.9204,C -2.0597,E1 24.8855,E2 225.4729} C_DIS
LIN {X -58.8584,Y -60.9629,Z 87,A -138.4646,B 24.9213,C -2.0491,E1 24.8897,E2 223.3421} C_DIS
LIN {X -56.8456,Y -62.8454,Z 87,A -136.4178,B 24.9211,C -2.0506,E1 24.8939,E2 221.2834} C_DIS
LIN {X -54.5873,Y -64.8169,Z 87,A -134.0132,B 24.9206,C -2.0578,E1 24.8991,E2 218.8524} C_DIS
LIN {X -49.616,Y -68.6969,Z 87,A -129.9584,B 24.9216,C -2.0442,E1 24.9081,E2 214.8155} C_DIS
LIN {X -44.6335,Y -72.0328,Z 87,A -125.9728,B 24.9223,C -2.0358,E1 24.9174,E2 210.8367} C_DIS
LIN {X -41.4006,Y -73.9377,Z 87,A -122.641,B 24.9207,C -2.056,E1 24.9257,E2 207.447} C_DIS
LIN {X -37.5403,Y -75.9705,Z 87,A -120.5198,B 24.9229,C -2.0275,E1 24.9308,E2 205.3879} C_DIS
LIN {X -34.9987,Y -77.1745,Z 87,A -118.7927,B 24.9235,C -2.0202,E1 24.9351,E2 203.6741} C_DIS
LIN {X -31.3363,Y -78.7335,Z 87,A -115.9521,B 24.9233,C -2.0219,E1 24.9425,E2 200.823} C_DIS
LIN {X -28.2757,Y -79.8831,Z 87,A -113.8589,B 24.9238,C -2.0164,E1 24.948,E2 198.7386} C_DIS
LIN {X -23.7163,Y -81.354,Z 87,A -110.4398,B 24.9235,C -2.0195,E1 24.9571,E2 195.3063} C_DIS
LIN {X -20.4777,Y -82.229,Z 87,A -108.1802,B 24.9236,C -2.0179,E1 24.9632,E2 193.047} C_DIS
LIN {X -15.9591,Y -83.2231,Z 87,A -105.3444,B 24.9244,C -2.0076,E1 24.9709,E2 190.2323} C_DIS
LIN {X -10.7678,Y -84.0527,Z 87,A -101.8441,B 24.9246,C -2.0049,E1 24.9806,E2 186.7352} C_DIS
LIN {X -5.0676,Y -84.5887,Z 87,A -97.2681,B 24.923,C -2.0266,E1 24.9934,E2 182.1057} C_DIS
LIN {X 0.2114,Y -84.7398,Z 87,A -93.6079,B 24.9227,C -2.0301,E1 25.0037,E2 178.4371} C_DIS
LIN {X 0.2114,Y -84.7398,Z 87,A -93.6079,B 24.9227,C -2.0301,E1 25.0037,E2 178.4371} C_DIS
Enddeposition()
LIN {X 0.5343,Y -83.8393,Z 87,A -94.3998,B 24.9239,C -2.0142,E1 25.0014,E2 179.2668} C_DIS
Startdeposition()
$VEL.CP = VEL_PRINT
LIN {X -3.9184,Y -83.7543,Z 87,A -97.9011,B 24.925,C -1.9996,E1 24.9915,E2 182.8029} C_DIS
LIN {X -7.7671,Y -83.485,Z 87,A -100.4999,B 24.925,C -2.0008,E1 24.9843,E2 185.3999} C_DIS
LIN {X -10.9838,Y -83.1232,Z 87,A -103.4075,B 24.9265,C -1.9804,E1 24.9761,E2 188.358} C_DIS
LIN {X -14.4559,Y -82.5908,Z 87,A -105.157,B 24.925,C -2.0005,E1 24.9714,E2 190.0617} C_DIS
LIN {X -17.9206,Y -81.908,Z 87,A -107.5213,B 24.9248,C -2.0029,E1 24.9649,E2 192.4228} C_DIS
LIN {X -21.352,Y -81.0827,Z 87,A -110.0278,B 24.9248,C -2.0014,E1 24.9581,E2 194.9365} C_DIS
LIN {X -24.0685,Y -80.317,Z 87,A -112.2153,B 24.9254,C -1.9952,E1 24.9522,E2 197.1425} C_DIS
LIN {X -27.8809,Y -79.0743,Z 87,A -115.0933,B 24.9254,C -1.9934,E1 24.9446,E2 200.0301} C_DIS
LIN {X -32.1495,Y -77.4382,Z 87,A -117.929,B 24.9246,C -2.0048,E1 24.9373,E2 202.845} C_DIS
LIN {X -34.8456,Y -76.263,Z 87,A -119.9366,B 24.9245,C -2.007,E1 24.9321,E2 204.8521} C_DIS
LIN {X -37.8599,Y -74.8118,Z 87,A -122.5892,B 24.9251,C -1.9993,E1 24.9255,E2 207.5301} C_DIS
LIN {X -42.5067,Y -72.2722,Z 87,A -126.219,B 24.9247,C -2.004,E1 24.9167,E2 211.1594} C_DIS
LIN {X -47.7391,Y -68.928,Z 87,A -129.9975,B 24.9232,C -2.0238,E1 24.9079,E2 214.9031} C_DIS
LIN {X -50.5838,Y -66.8678,Z 87,A -132.6689,B 24.9235,C -2.0203,E1 24.9019,E2 217.5923} C_DIS
LIN {X -54.3634,Y -63.8333,Z 87,A -135.5509,B 24.9221,C -2.0385,E1 24.8957,E2 220.4418} C_DIS
LIN {X -55.8008,Y -62.5809,Z 87,A -137.1122,B 24.9224,C -2.0338,E1 24.8924,E2 222.0205} C_DIS
LIN {X -58.3923,Y -60.1705,Z 87,A -139.4639,B 24.9219,C -2.0406,E1 24.8877,E2 224.3658} C_DIS
LIN {X -60.6705,Y -57.8736,Z 87,A -141.8868,B 24.922,C -2.0394,E1 24.8829,E2 226.8019} C_DIS
LIN {X -63.4211,Y -54.8452,Z 87,A -144.7112,B 24.9216,C -2.0449,E1 24.8777,E2 229.626} C_DIS
LIN {X -66.0318,Y -51.6723,Z 87,A -147.8268,B 24.9217,C -2.0431,E1 24.8722,E2 232.7605} C_DIS
LIN {X -68.5751,Y -48.2468,Z 87,A -150.3218,B 24.9203,C -2.0617,E1 24.8682,E2 235.2231} C_DIS
LIN {X -70.2048,Y -45.8421,Z 87,A -152.2385,B 24.9198,C -2.0686,E1 24.8653,E2 237.133} C_DIS
LIN {X -71.7439,Y -43.3926,Z 87,A -155.1095,B 24.9212,C -2.0496,E1 24.861,E2 240.0641} C_DIS
LIN {X -73.8104,Y -39.7762,Z 87,A -156.9004,B 24.9184,C -2.0857,E1 24.8587,E2 241.7781} C_DIS
Enddeposition()
END
